// TIA Portal project "TestProject" (V19)

(* hardware
DEVICE "S7-1500/ET200MP station_3"  S7-1500 station
   slot 0: "Rail_0"  Rack  6ES7 590-1***0-0AA0
   slot 1: "PLC_3"  CPU 1511-1 PN  6ES7 511-1AK02-0AB0  V2.8
      slot 3: "CPU display_1"  6ES7591-1AA00-0AA0
      slot 32768: "PROFINET interface_1"  X1
         slot 32769: "Port_1"  X1 P1
         slot 32770: "Port_2"  X1 P2
      slot 34817: "Virtual CP interface port_1"  Virtual CP interface port  Virtual CP interface port
*)

// ===== PLC "PLC_3"  CPU 1511-1 PN =====

DATA_BLOCK "DTLToString_ISO_DB"   // DB1
{ S7_Optimized_Access := 'TRUE' }
VERSION : 0.1
   VAR
      "date" : DTL;
      separator : Char;
      DTLToString_ISO : String;
   END_VAR
BEGIN
END_DATA_BLOCK

DATA_BLOCK "ExtractStringFromCharArray_DB"   // DB2
{ S7_Optimized_Access := 'TRUE' }
VERSION : 0.1
   VAR
      textBefore : String;
      textAfter : String;
      extractedString : String;
      status : Word;
      searchIn : Array[0..9] of Char;
      ExtractStringFromCharArray : Word;
   END_VAR
BEGIN
END_DATA_BLOCK

DATA_BLOCK "MatrixAddition_DB"   // DB3
{ S7_Optimized_Access := 'TRUE' }
VERSION : 0.1
   VAR
      matrix1 : Array[1..2, 1..2] of LReal;
      matrix2 : Array[1..2, 1..2] of LReal;
      error : Bool;
      status : Word;
      matrixResult : Array[1..2, 1..2] of LReal;
   END_VAR
BEGIN
END_DATA_BLOCK

DATA_BLOCK "RandomRange_DInt_DB"   // DB4
{ S7_Optimized_Access := 'TRUE' }
VERSION : 0.1
   VAR
      minValue : DInt;
      maxValue : DInt;
      error : Bool;
      status : Word;
      subfunctionStatus : Word;
      RandomRange_DInt : DInt;
   END_VAR
BEGIN
END_DATA_BLOCK

DATA_BLOCK "SearchMinMax_DInt_DB"   // DB5
{ S7_Optimized_Access := 'TRUE' }
VERSION : 0.1
   VAR
      values : Array[0..9] of DInt;
      minValue : DInt;
      minValueIndex : DInt;
      maxValue : DInt;
      maxValueIndex : DInt;
   END_VAR
BEGIN
END_DATA_BLOCK

DATA_BLOCK "StringToTaddr_DB"   // DB6
{ S7_Optimized_Access := 'TRUE' }
VERSION : 0.1
   VAR
      ipAddressString : String;
      error : Bool;
      status : Word;
      StringToTaddr : TADDR_Param;
   END_VAR
BEGIN
END_DATA_BLOCK

DATA_BLOCK "FIFO_DB"   // DB7
{ S7_Optimized_Access := 'TRUE' }
VERSION : 0.1
// stored: InstanceOfName FIFO
"FIFO"
BEGIN
END_DATA_BLOCK

DATA_BLOCK "FIFO_DBG"   // DB8
{ S7_Optimized_Access := 'TRUE' }
VERSION : 0.1
   VAR
      enqueue : Bool;
      dequeue : Bool;
      reset : Bool;
      clear : Bool;
      initialItem : Int;
      error : Bool;
      status : Word;
      subFunctionStatus : Word;
      elementCount : DInt;
      isEmpty : Bool;
      item : Int;
      buffer : Array[1..3] of Int;
   END_VAR
BEGIN
END_DATA_BLOCK

DATA_BLOCK "FloatingAverage_DB"   // DB9
{ S7_Optimized_Access := 'TRUE' }
VERSION : 0.1
// stored: InstanceOfName FloatingAverage
"FloatingAverage"
BEGIN
END_DATA_BLOCK

DATA_BLOCK "Frequency_DB"   // DB10
{ S7_Optimized_Access := 'TRUE' }
VERSION : 0.1
// stored: InstanceOfName Frequency
"Frequency"
BEGIN
END_DATA_BLOCK

DATA_BLOCK "GetBitStates_DB"   // DB11
{ S7_Optimized_Access := 'TRUE' }
VERSION : 0.1
// stored: InstanceOfName GetBitStates
"GetBitStates"
BEGIN
END_DATA_BLOCK

DATA_BLOCK "Integration_DB"   // DB12
{ S7_Optimized_Access := 'TRUE' }
VERSION : 0.1
// stored: InstanceOfName Integration
"Integration"
BEGIN
END_DATA_BLOCK

DATA_BLOCK "ShellSort_DInt_DB"   // DB13
{ S7_Optimized_Access := 'TRUE' }
VERSION : 0.1
// stored: InstanceOfName ShellSort_DInt
"ShellSort_DInt"
BEGIN
END_DATA_BLOCK

DATA_BLOCK "ShellSort_DInt_DBG"   // DB14
{ S7_Optimized_Access := 'TRUE' }
VERSION : 0.1
   VAR
      sortDirection : Bool;
      error : Bool;
      status : Word;
      "array" : Array[1..5] of DInt;
   END_VAR
BEGIN
END_DATA_BLOCK

DATA_BLOCK "StackMin_DB"   // DB15
{ S7_Optimized_Access := 'TRUE' }
VERSION : 0.1
// stored: InstanceOfName StackMin
"StackMin"
BEGIN
END_DATA_BLOCK

DATA_BLOCK "StackMin_DBG"   // DB16
{ S7_Optimized_Access := 'TRUE' }
VERSION : 0.1
   VAR
      push : Bool;
      pop : Bool;
      reset : Bool;
      error : Bool;
      status : Word;
      item : Int;
      stack : Array[0..3] of Int;
   END_VAR
BEGIN
END_DATA_BLOCK

DATA_BLOCK "TempCtrl_DB"   // DB17
{ S7_Optimized_Access := 'TRUE' }
VERSION : 0.1
// stored: InstanceOfName TempCtrl
"TempCtrl"
BEGIN
END_DATA_BLOCK

DATA_BLOCK "LightsControl_DB"   // DB18
{ S7_Optimized_Access := 'TRUE' }
VERSION : 0.1
// stored: InstanceOfName LightsControl
"LightsControl"
BEGIN
END_DATA_BLOCK

DATA_BLOCK "MatrixAddition_DBG"   // DB19
{ S7_Optimized_Access := 'TRUE' }
VERSION : 0.1
   VAR
      matrix1 : Array[1..4] of LReal;
      matrix2 : Array[1..4] of LReal;
      matrixResult : Array[1..4] of LReal;
   END_VAR
BEGIN
END_DATA_BLOCK

DATA_BLOCK "MatrixMultiplication_DB"   // DB20
{ S7_Optimized_Access := 'TRUE' }
VERSION : 0.1
   VAR
      matrix1 : Array[1..2, 1..2] of LReal;
      matrix2 : Array[1..2, 1..2] of LReal;
      error : Bool;
      status : Word;
      matrixResult : Array[1..2, 1..2] of LReal;
   END_VAR
BEGIN
END_DATA_BLOCK

DATA_BLOCK "MatrixMultiplication_DBG"   // DB21
{ S7_Optimized_Access := 'TRUE' }
VERSION : 0.1
   VAR
      matrix1 : Array[1..4] of LReal;
      matrix2 : Array[1..4] of LReal;
      matrixResult : Array[1..4] of LReal;
   END_VAR
BEGIN
END_DATA_BLOCK

FUNCTION_BLOCK "FIFO"   // FB1, SCL
{ S7_Optimized_Access := 'TRUE' }
   VAR_INPUT
      enqueue : Bool := FALSE;
      dequeue : Bool := FALSE;
      reset : Bool;
      clear : Bool;
      initialItem : Variant;
   END_VAR
   VAR_OUTPUT
      error : Bool;
      status : Word;
      elementCount : DInt := 0;
      isEmpty : Bool := FALSE;
   END_VAR
   VAR_IN_OUT
      item : Variant;
      buffer : Variant;
   END_VAR
   VAR
      statEdgesMem : Struct
         enqueue : Bool;
         dequeue : Bool;
         clear : Bool;
      END_STRUCT;
      statFirstItemIndex : Int := -1;
      statNextEmptyItemIndex : Int := 0;
      statElementCount : DInt;
   END_VAR
   VAR_TEMP
      tempEdges : Struct
         enqueue : Bool;
         dequeue : Bool;
         clear : Bool;
      END_STRUCT;
      tempInternalError : Int;
      tempNewFirstItemIndex : Int;
      tempNewNextEmptyItemIndex : Int;
      tempBufferSize : UDInt;
      tempCounter : Int;
   END_VAR
   VAR CONSTANT
      BUFFER_IS_EMPTY : Int := -1;
      NO_INTERNAL_ERROR : Int := 0;
      BUFFER_INITIALIZED : Int := -1;
      EMPTY_INITIALIZED : Int := 0;
      INDEX_BEGINNING : Int := 0;
      COUNT_ELEMENTS : UDInt := 1;
      INCREMENT : Int := 1;
      BUFFER_SIZE_CORRECTION : UDInt := 1;
      COUNTER_LOWER_LIMIT : Int := 0;
      ZERO_ELEMENTS : DInt := 0;
      STATUS_NO_ERROR : Word := 16#0000;
      STATUS_NO_CURRENT_JOBS : Word := 16#7000;
      ERR_BUFFER_EMPTY : Word := 16#8001;
      ERR_BUFFER_FULL : Word := 16#8002;
      ERR_NO_ARRAY : Word := 16#8200;
      ERR_WRONG_TYPE_ITEM : Word := 16#8201;
      ERR_WRONG_TYPE_INITIAL_ITEM : Word := 16#8202;
      ERR_INDEX_IN_ARRAY_LIMITS_1 : Word := 16#8601;
      ERR_INDEX_IN_ARRAY_LIMITS_2 : Word := 16#8602;
      ERR_CLEAR_BUFFER : Word := 16#8610;
      ERR_RETURN_FIRST_ENTRY : Word := 16#8611;
      ERR_REPLACE_ITEM_BY_INIT_VALUE : Word := 16#8612;
      ERR_WRITE_ENTRY : Word := 16#8613;
   END_VAR
BEGIN
   REGION Block info header
       //===============================================================================
       // Title:           FIFO
       // Comment/Function: FIFO (First In First Out)
       //                   Queue / ring buffer memory

       //=============================================================================
   END_REGION Block info header

   REGION Block execution control
       // collect edges
       #tempEdges.enqueue := #enqueue AND NOT #statEdgesMem.enqueue;
       #tempEdges.dequeue := #dequeue AND NOT #statEdgesMem.dequeue;
       #tempEdges.clear := #clear AND NOT #statEdgesMem.clear;
       // store values for edge detection
       #statEdgesMem.enqueue := #enqueue;
       #statEdgesMem.dequeue := #dequeue;
       #statEdgesMem.clear := #clear;

       // This program code section is only executed if no trigger input is active
       IF NOT (#enqueue OR #dequeue OR #reset OR #clear) THEN
           // If an error occurred during program execution,
           // the status "No Current Job" is used 16#7000 afterwarts when the triggers are reseted
           #error := false;
           #status := #STATUS_NO_CURRENT_JOBS;

           // the program processing OF the FB is terminated
           RETURN;
       END_IF;
   END_REGION

   REGION Validation of inputs
       // check whether the ring #buffer is an ARRAY.
       // IF so, the number OF the ARRAY elements is read out.
       // IF it is NOT an ARRAY, the program execution is terminated at this point
       IF IS_ARRAY(#buffer) THEN
           #tempBufferSize := CountOfElements(#buffer);
       ELSE
           #error := true;
           #status := #ERR_NO_ARRAY;

           RETURN;
       END_IF;

       // check whether the data type OF the ARRAY elements matches
       // the data type OF the entry (#item). IF the data types DO NOT match,
       // the program execution is terminated at this point
       IF (TypeOf(#item) <> TypeOfElements(#buffer)) THEN
           #error := true;
           #status := #ERR_WRONG_TYPE_ITEM;

           RETURN;
       END_IF;

       // check whether the initial value OF the ring #buffer
       // matches the entry (tag #item). IF the data types DO NOT match,
       // the program execution is terminated at this point
       IF (TypeOf(#item) <> TypeOf(#initialItem)) THEN
           #error := true;
           #status := #ERR_WRONG_TYPE_INITIAL_ITEM;

           RETURN;
       END_IF;

       // check whether the variable indices are within the ARRAY limits.
       // IF they are NOT, the program execution is terminated at this point
       IF (#statNextEmptyItemIndex >= #tempBufferSize) THEN
           #error := true;
           #status := #ERR_INDEX_IN_ARRAY_LIMITS_1;

           RETURN;
       ELSIF (#statFirstItemIndex >= #tempBufferSize) THEN
           #error := true;
           #status := #ERR_INDEX_IN_ARRAY_LIMITS_2;

           RETURN;
       END_IF;

       // If resetBuffer is "TRUE", the buffer counters are reset
       IF #reset THEN
           #statFirstItemIndex := #BUFFER_INITIALIZED;
           #statNextEmptyItemIndex := #EMPTY_INITIALIZED;
           #statElementCount := #EMPTY_INITIALIZED;
           #elementCount := #EMPTY_INITIALIZED;
           #isEmpty := true;
           RETURN;
       END_IF;

       // If clearBuffer has rising edge, the buffer is initialized by initial values
       IF #tempEdges.clear THEN
           FOR #tempCounter := #COUNTER_LOWER_LIMIT TO UDINT_TO_INT(#tempBufferSize - #BUFFER_SIZE_CORRECTION) DO

               #tempInternalError := MOVE_BLK_VARIANT(SRC := #initialItem,
                                                      COUNT := #COUNT_ELEMENTS,
                                                      SRC_INDEX := #INDEX_BEGINNING,
                                                      DEST_INDEX := #tempCounter,
                                                      DEST => #buffer);
           END_FOR;

           // checks whether a local error has occurred.
           IF (#tempInternalError <> #NO_INTERNAL_ERROR) THEN
               #error := true;
               #status := #ERR_CLEAR_BUFFER;

           END_IF;

           // reset counters
           #statFirstItemIndex := #BUFFER_INITIALIZED;
           #statNextEmptyItemIndex := #EMPTY_INITIALIZED;
           #statElementCount := #EMPTY_INITIALIZED;
           #elementCount := #EMPTY_INITIALIZED;
           #isEmpty := true;
           RETURN;
       END_IF;
   END_REGION

   REGION FIFO algorithm  
       IF #tempEdges.dequeue THEN
           REGION dequeue
               // check whether the ring #buffer is empty
               // IF this is the CASE, program execution is terminated at this point
               IF (#statFirstItemIndex = #BUFFER_IS_EMPTY) THEN
                   #error := true;
                   #status := #ERR_BUFFER_EMPTY;

                   RETURN;
               END_IF;

               // return the first entry of the ring buffer
               #tempInternalError := MOVE_BLK_VARIANT(SRC := #buffer,
                                                      COUNT := #COUNT_ELEMENTS,
                                                      SRC_INDEX := #statFirstItemIndex,
                                                      DEST_INDEX := #INDEX_BEGINNING,
                                                      DEST => #item);

               // check whether a local error has occurred
               IF (#tempInternalError <> #NO_INTERNAL_ERROR) THEN
                   #error := true;
                   #status := #ERR_RETURN_FIRST_ENTRY;

                   RETURN;
               END_IF;

               // check whether the ring #buffer contains ARRAY elements
               // IF it does, the first entry is passed further on and the index is incremented BY 1
               #tempInternalError := MOVE_BLK_VARIANT(SRC := #initialItem,
                                                      COUNT := #COUNT_ELEMENTS,
                                                      SRC_INDEX := #INDEX_BEGINNING,
                                                      DEST_INDEX := #statFirstItemIndex,
                                                      DEST => #buffer);

               // check whether a local error has occurred
               IF (#tempInternalError <> #NO_INTERNAL_ERROR) THEN
                   #error := true;
                   #status := #ERR_REPLACE_ITEM_BY_INIT_VALUE;

                   RETURN;
               END_IF;

               // calculate the new index of the first entry
               #tempNewFirstItemIndex := #statFirstItemIndex + #INCREMENT;
               #tempNewFirstItemIndex := #tempNewFirstItemIndex MOD UDINT_TO_INT(#tempBufferSize);

               // check whether the ring buffer is empty
               IF (#statNextEmptyItemIndex = #tempNewFirstItemIndex) THEN
                   // If the ring buffer is empty, the index is set to 0
                   #statFirstItemIndex := #BUFFER_INITIALIZED;
                   #statNextEmptyItemIndex := #EMPTY_INITIALIZED;
               ELSE
                   // The index of the first entry is changed
                   #statFirstItemIndex := #tempNewFirstItemIndex;
               END_IF;

               // Evaluation of the number of elements in the stack
               #statElementCount -= #INCREMENT;

           END_REGION dequeue

       ELSIF #tempEdges.enqueue THEN
           REGION enqueue
               // check whether the ring #buffer is full
               // IF this is the CASE, program execution is terminated at this point
               IF (#statNextEmptyItemIndex = #statFirstItemIndex) THEN
                   #error := true;
                   #status := #ERR_BUFFER_FULL;

                   RETURN;
               END_IF;

               // write the entry to the ring buffer
               #tempInternalError := MOVE_BLK_VARIANT(SRC := #item,
                                                      COUNT := #COUNT_ELEMENTS,
                                                      SRC_INDEX := #INDEX_BEGINNING,
                                                      DEST_INDEX := #statNextEmptyItemIndex,
                                                      DEST => #buffer);

               // check whether a local error has occurred
               IF (#tempInternalError <> #NO_INTERNAL_ERROR) THEN
                   #error := true;
                   #status := #ERR_WRITE_ENTRY;

                   RETURN;
               END_IF;

               // increment the index by 1 and calculates the new empty entry index
               #tempNewNextEmptyItemIndex := (#statNextEmptyItemIndex + #INCREMENT) MOD UDINT_TO_INT(#tempBufferSize);
               #statNextEmptyItemIndex := #tempNewNextEmptyItemIndex;

               // check which index the "#firstItemIndex" tag has
               // IF the number = -1, the ring buffer is initialized
               // AND the entry is written TO the ring #buffer
               // Therefore, "0" must be assigned TO the tag
               IF (#statFirstItemIndex = #BUFFER_INITIALIZED) THEN
                   #statFirstItemIndex := #INDEX_BEGINNING;
               END_IF;

               // Evaluation of the number of elements in the stack
               #statElementCount += #INCREMENT;
           END_REGION enqueue
       END_IF;
   END_REGION

   REGION Writing to outputs
       #elementCount := #statElementCount;
       #isEmpty := #statElementCount <= #ZERO_ELEMENTS;

       #error := false;
       #status := #STATUS_NO_ERROR;

       // no error handling by ENO needed
       ENO := TRUE;
   END_REGION
END_FUNCTION_BLOCK

FUNCTION_BLOCK "FloatingAverage"   // FB2, SCL
{ S7_Optimized_Access := 'TRUE' }
   VAR_INPUT
      cyclicExecution : Bool := FALSE;
      trigger : Bool;
      value : LReal;
      windowSize : Int := 100;
      reset : Bool;
   END_VAR
   VAR_OUTPUT
      average : LReal;
      windowSizeReached : Bool;
      error : Bool;
      status : Word;
   END_VAR
   VAR
      statValues : Array[#ZERO_INT..#MAX_WINDOW_SIZE] of LReal;
      statValuesSum : LReal := 0.0;
      statArithmeticAverage : LReal := 0.0;
      statWindowSizeOld : Int := 0;
      statCounter : Int := 0;
      statwindowSizeReached : Bool;
      statTriggerOld : Bool := FALSE;
   END_VAR
   VAR_TEMP
      tempValue : LReal;
      tempIndex : Int;
      tempTriggerEdge : Bool;
   END_VAR
   VAR CONSTANT
      ZERO_INT : Int := 0;
      ZERO_LREAL : LReal := 0.0;
      MAX_WINDOW_SIZE : Int := 100;
      INCREMENT : Int := 1;
      STATUS_FINISHED_NO_ERROR : Word := 16#0000;
      ERR_WRONG_WINDOW_SIZE : Word := 16#8200;
   END_VAR
BEGIN
   REGION Block info header
       //===============================================================================
       // Title:            FloatingAverage
       // Comment/Function: This function block calculates the floating arithmetic average
       //                   of incoming REAL values each cycle or each trigger impulse.

       //=============================================================================
   END_REGION Block info header

   REGION DESCRIPTION
       (/**/)
   END_REGION DESCRIPTION

   REGION Initialization and input data processing
       // Copy commonly used data to temp variables
       #tempValue := #value;

       // Positive edge detection for triggering of calculation
       #tempTriggerEdge := #trigger AND NOT #statTriggerOld;
       #statTriggerOld := #trigger;

       // Reset OR if window size changes the calculation
       IF #reset OR (#windowSize <> #statWindowSizeOld) THEN
           #statWindowSizeOld := #windowSize;
           #statCounter := #ZERO_INT;
           #statValuesSum := #ZERO_LREAL;
           #statArithmeticAverage := #ZERO_LREAL;
           #average := #ZERO_LREAL;
           #windowSizeReached := FALSE;
           #statwindowSizeReached := FALSE;
           #error := false;
           #status := #STATUS_FINISHED_NO_ERROR;
           RETURN;

           // Check window size, in case of incorrect window size setup an error
       ELSIF (#windowSize <= #ZERO_INT) OR (#windowSize > #MAX_WINDOW_SIZE) THEN
           #statWindowSizeOld := #windowSize;
           #statCounter := #ZERO_INT;
           #statValuesSum := #ZERO_LREAL;
           #statArithmeticAverage := #ZERO_LREAL;
           #average := #ZERO_LREAL;
           #statwindowSizeReached := FALSE;
           #windowSizeReached := FALSE;
           #error := TRUE;
           #status := #ERR_WRONG_WINDOW_SIZE; // Info "No correct set of window size"
           RETURN;
       END_IF;
   END_REGION

   REGION Floating average calculation
       // Triggered calculation OR cyclicly operation
       IF #cyclicExecution OR #tempTriggerEdge THEN

           //Calculate array counter by using modulo
           #tempIndex := #statCounter MOD #windowSize;

           // First step - fill the Array with values
           // as long as desired window size is not reached
           // counter and array starts with zero
           IF (#statCounter < #windowSize) THEN
               // Add value to sum
               #statValuesSum += #tempValue;
               // Add value to window
               #statValues[#tempIndex] := #tempValue;
               // Increment counter
               #statCounter += #INCREMENT;
               // Calculate avarage value
               #statArithmeticAverage := #statValuesSum / #statCounter;

           ELSE
               // wuindow size is reached, set output
               #statwindowSizeReached := TRUE;
               // Add value to sum
               #statValuesSum += #tempValue - #statValues[#tempIndex];
               // Add value to window
               #statValues[#tempIndex] := #tempValue;
               // Calculate avarage value
               #statArithmeticAverage := #statValuesSum / #windowSize;

               // Manipulate counter value of window if modulo calc result is zero
               IF (#tempIndex = #ZERO_INT) THEN
                   #statCounter := #windowSize + #INCREMENT;
               ELSE
                   // Increment counter
                   #statCounter += #INCREMENT;
               END_IF;
           END_IF;
       END_IF;
   END_REGION

   REGION Outputs
       #average := #statArithmeticAverage;
       #windowSizeReached := #statwindowSizeReached;
       #error := FALSE;
       #status := #STATUS_FINISHED_NO_ERROR;

       // ENO mechanism is not used - forced to true
       ENO := TRUE;
   END_REGION
END_FUNCTION_BLOCK

FUNCTION_BLOCK "Frequency"   // FB3, SCL
{ S7_Optimized_Access := 'TRUE' }
   VAR_INPUT
      frequency : Real := 0.0;
      pulsePauseRatio : Real := 1.0;
   END_VAR
   VAR_OUTPUT
      clock : Bool;
      countdown : Time;
   END_VAR
   VAR
      instTofTimePulse : TOF_TIME;
      instTofTimePause : TOF_TIME;
      statFrequencyOld : Real;
      statPulsePauseRatioOld : Real;
      statTimePulse : Time;
      statTimePause : Time;
   END_VAR
   VAR_TEMP
      tempPulseRate : Real;
      tempPauseRate : Real;
      tempCountdown : Time;
   END_VAR
   VAR CONSTANT
      ZERO : Real := 0.0;
      ZERO_TIME : Time := T#0MS;
      SECOND_IN_MS : Real := 1000.0;
      ONE : Real := 1.0;
   END_VAR
BEGIN
   REGION Block info header
       //=============================================================================
       // Title:            Frequency
       // Comment/Function: This function generates a signal that changes between the values `FALSE` and `TRUE` depending on a defined frequency and a pulse pause ratio.

       //=============================================================================
   END_REGION Block info header

   REGION Calculation of settings and program execution
       // If input <= 0.0 the block is disabled
       IF (#frequency <= #ZERO) OR (#pulsePauseRatio <= #ZERO) THEN
           #clock := FALSE;
           #tempCountdown := #ZERO_TIME;
       ELSE

           //Calculating function frequency and pulse pause ratio only when an input is changed
           IF #statFrequencyOld <> #frequency OR #statPulsePauseRatioOld <> #pulsePauseRatio THEN
               RESET_TIMER(TIMER := #instTofTimePause);
               RESET_TIMER(TIMER := #instTofTimePulse);

               #tempPulseRate := #pulsePauseRatio / (#pulsePauseRatio + #ONE); // Calculate pulse rate   
               #tempPauseRate := #ONE - #tempPulseRate;                      // Calculate pause rate   
               #statTimePulse := UDINT_TO_TIME(REAL_TO_UDINT((#SECOND_IN_MS * #tempPulseRate / #frequency))); // Calculate pulse time   
               #statTimePause := UDINT_TO_TIME(REAL_TO_UDINT((#SECOND_IN_MS * #tempPauseRate / #frequency))); // Calculate pause time
               #statFrequencyOld := #frequency;
               #statPulsePauseRatioOld := #pulsePauseRatio;
           END_IF;

           //Two time off-delay timers that are resetting each other on expiration
           #instTofTimePulse(IN := NOT #instTofTimePause.Q,
                             PT := #statTimePulse);

           //If timer for pulse is running, remaining time of the PULSE is calculated
           #tempCountdown := #statTimePulse - #instTofTimePulse.ET;

           #instTofTimePause(IN := #instTofTimePulse.Q,
                             PT := #statTimePause);

           //If timer for pulse is NOT running, remaining time of the PAUSE is calculated
           IF #tempCountdown = #ZERO_TIME THEN
               #tempCountdown := #statTimePause - #instTofTimePause.ET;
           END_IF;

       END_IF;
   END_REGION

   REGION Writing to outputs
       // Assigning value of the pulse timer to the clock output
       #clock := #instTofTimePulse.Q;
       #countdown := #tempCountdown;
       //ENO mechanism is not used - forced to true.
       ENO := TRUE;
   END_REGION
END_FUNCTION_BLOCK

FUNCTION_BLOCK "GetBitStates"   // FB4, SCL
{ S7_Optimized_Access := 'TRUE' }
   VAR_INPUT
      value : DWord;
   END_VAR
   VAR_OUTPUT
      hasChanged : Bool;
      hasRisingEdges : Bool;
      risingBits : DWord;
      noOfRisingBits : USInt;
      hasFallingEdges : Bool;
      fallingBits : DWord;
      noOfFallingBits : USInt;
   END_VAR
   VAR
      statPreviousValue : DWord;
   END_VAR
   VAR_TEMP
      tempRisingResult : DWord;
      tempNoRisingBits : DWord;
      tempFallingResult : DWord;
      tempNoFallingBits : DWord;
   END_VAR
   VAR CONSTANT
      ZERO_EDGES : DWord;
   END_VAR
BEGIN
   REGION BLOCK INFO HEADER
       //============================================================================
       // Title:            GetBitStates
       // Comment/Function: Check DWord for edges, falling as well as rising.  
       //                   Returns the number of edges, DWords with edge bits and a bool if edge(s) exists.
       //                   https://graphics.stanford.edu/~seander/bithacks.html#CountBitsSetParallel

       //=============================================================================
   END_REGION BLOCK INFO HEADER

   REGION PROGRAM LOGIC
       // Get edges from input DWord and DWord from previous cycle
       #tempRisingResult := #value AND NOT #statPreviousValue;
       #tempFallingResult := NOT #value AND #statPreviousValue;

       // Store value for next cycle
       #statPreviousValue := #value;

       // Copy edge result into work variable for counting the number of rising edges
       #tempNoRisingBits := #tempRisingResult;
       // Count number of rising edges, algorythm descriped from: https://graphics.stanford.edu/~seander/bithacks.html#CountBitsSetParallel
       #tempNoRisingBits := UDINT_TO_DWORD(DWORD_TO_UDINT(#tempNoRisingBits) - DWORD_TO_UDINT(SHR(IN := #tempNoRisingBits, N := 1) AND 16#55555555));
       #tempNoRisingBits := UDINT_TO_DWORD(DWORD_TO_UDINT(#tempNoRisingBits & 16#33333333) + DWORD_TO_UDINT(SHR(IN := #tempNoRisingBits, N := 2) AND 16#33333333));
       #tempNoRisingBits := SHR(IN := UDINT_TO_DWORD(DWORD_TO_UDINT(UDINT_TO_DWORD(DWORD_TO_UDINT(#tempNoRisingBits) + DWORD_TO_UDINT(SHR(IN := #tempNoRisingBits, N := 4))) AND 16#0F0F0F0F) * DWORD_TO_UDINT(16#01010101)), N := 24);

       // Copy edges result into work variable for counting the number of falling edges
       #tempNoFallingBits := #tempFallingResult;
       // Count number of falling edges, algorythm descriped from: https://graphics.stanford.edu/~seander/bithacks.html#CountBitsSetParallel
       #tempNoFallingBits := UDINT_TO_DWORD(DWORD_TO_UDINT(#tempNoFallingBits) - DWORD_TO_UDINT(SHR(IN := #tempNoFallingBits, N := 1) AND 16#55555555));
       #tempNoFallingBits := UDINT_TO_DWORD(DWORD_TO_UDINT(#tempNoFallingBits & 16#33333333) + DWORD_TO_UDINT(SHR(IN := #tempNoFallingBits, N := 2) AND 16#33333333));
       #tempNoFallingBits := SHR(IN := UDINT_TO_DWORD(DWORD_TO_UDINT(UDINT_TO_DWORD(DWORD_TO_UDINT(#tempNoFallingBits) + DWORD_TO_UDINT(SHR(IN := #tempNoFallingBits, N := 4))) AND 16#0F0F0F0F) * DWORD_TO_UDINT(16#01010101)), N := 24);
   END_REGION PROGRAM LOGIC

   REGION OUTPUTS
       #hasChanged := (#tempRisingResult > #ZERO_EDGES) OR (#tempFallingResult > #ZERO_EDGES);
       #hasRisingEdges := #tempRisingResult > #ZERO_EDGES;
       #risingBits := #tempRisingResult;
       #noOfRisingBits := DWORD_TO_USINT(#tempNoRisingBits);

       #hasFallingEdges := #tempFallingResult > #ZERO_EDGES;
       #fallingBits := #tempFallingResult;
       #noOfFallingBits := DWORD_TO_USINT(#tempNoFallingBits);

       // ENO not needed, no error evaluation needed
       ENO := FALSE;
   END_REGION OUTPUTS
END_FUNCTION_BLOCK

FUNCTION_BLOCK "Integration"   // FB5, SCL
{ S7_Optimized_Access := 'TRUE' }
   VAR_INPUT
      enable : Bool;
      value : LReal;
      reset : Bool;
   END_VAR
   VAR_OUTPUT
      integral : LReal;
      error : Bool;
      status : Word;
   END_VAR
   VAR
      statLastTime : DTL;
      statInputOldValue : LReal;
      statIntegral : LReal;
   END_VAR
   VAR_TEMP
      tempSysTime : DTL;
      tempTimeDiffrence : LReal;
      tempCalculation : LReal;
      tempRetval : Word;
   END_VAR
   VAR CONSTANT
      CLEAR_TIME : DTL;
      SECOND_IN_MS : LReal := 1000.0;
      DIVIDE_BY_TWO : LReal := 2.0;
      ZERO : LReal := 0.0;
      STATUS_EXECUTION_FINISHED_NO_ERROR : Word := 16#0000;
      SUB_STATUS_NO_ERROR : Word := 16#0000;
      ERR_READ_SYS_TIME : Word := 16#8600;
   END_VAR
BEGIN
   REGION Block info header
       //============================================================================
       // Title:            Integration
       // Comment/Function: Integrates the input value
       //                   integration by trapezoidal rule

       //=============================================================================
   END_REGION Block info header

   //Reset region must be before the enable region so that even if the function disabled, the user can reset the values.
   REGION Reset the function
       IF #reset THEN
           #statInputOldValue := #ZERO;
           #statIntegral := #ZERO;

           // Clear LastTime value.
           // Initial condition - first Delta time will be 0.
           #statLastTime := #CLEAR_TIME;

           #integral := #ZERO;
           #error := false;
           #status := #STATUS_EXECUTION_FINISHED_NO_ERROR;

           RETURN;
       END_IF;
   END_REGION Reset the function

   REGION Enable/Disable integral calculation
       IF NOT #enable THEN
           #statInputOldValue := #ZERO;

           // Clear LastTime value.
           // If it is not cleared when the function is enabled again,
           // the first value will be multiplied with the time difference of the whole disable time
           // Initial condition - first Delta time will be 0.
           #statLastTime := #CLEAR_TIME;

           #integral := #statIntegral;
           #error := false;
           #status := #STATUS_EXECUTION_FINISHED_NO_ERROR;

           RETURN;
       END_IF;
   END_REGION Enable/Disable integral calculation

   REGION Get system time
       // Read system time
       #tempRetval := INT_TO_WORD(RD_SYS_T(OUT => #tempSysTime));

       // Error Handling read system time
       IF (#tempRetval > #SUB_STATUS_NO_ERROR) THEN
           #integral := #statIntegral;
           #error := TRUE;
           #status := #ERR_READ_SYS_TIME;

           RETURN;
       END_IF;
   END_REGION

   REGION Calculating the integral
       // Calculate time difference between last and actual time
       // coverting from DTL via time and DInt to Real
       // scale from millisecond to second
       #tempTimeDiffrence := DINT_TO_REAL(TIME_TO_DINT(T_DIFF(IN1 := #tempSysTime, IN2 := #statLastTime))) / #SECOND_IN_MS;

       // Write actual to last time
       #statLastTime := #tempSysTime;

       // integration by trapezoidal rule
       // add LastScalIn to ScalIn
       // divide by two --> avarage of both - old and actual value
       // multiply with time delta --> area unterneath the both borders
       #tempCalculation := (#value + #statInputOldValue) * #tempTimeDiffrence / #DIVIDE_BY_TWO;

       // Calculate new integral
       #statIntegral += #tempCalculation;

       // Save last input
       #statInputOldValue := #value;
   END_REGION Calculating the integral

   REGION Write outputs
       #integral := #statIntegral;
       #error := false;
       #status := #STATUS_EXECUTION_FINISHED_NO_ERROR;


       //ENO mechanism is not used
       ENO := TRUE;
   END_REGION Write outputs
END_FUNCTION_BLOCK

FUNCTION_BLOCK "ShellSort_DInt"   // FB6, SCL
{ S7_Optimized_Access := 'TRUE' }
   VAR_INPUT
      sortDirection : Bool;
   END_VAR
   VAR_OUTPUT
      error : Bool;
      status : Word;
   END_VAR
   VAR_IN_OUT
      "array" : Array[*] of DInt;
   END_VAR
   VAR
      tempArray : Array[1..#MAX_ARRAY_ELEMENTS] of DInt;
   END_VAR
   VAR_TEMP
      tempLowerLimit : DInt;
      tempUpperLimit : DInt;
      tempNoOfElements : DInt;
      tempGap : DInt;
      tempLoopIndex : DInt;
      tempExchangeIndex : DInt;
      tempExchangeVariable : DInt;
      tempArrayOffset : DInt;
   END_VAR
   VAR CONSTANT
      ARRAY_FIRST_DIMENSION : UInt := 1;
      ARRAY_START_INDEX : UInt := 1;
      SINGLE_ARRAY_ELEMENT : DInt := 1;
      GAP_INIT : Int := 1;
      GAP_THRESHOLD : Int := 1;
      GAP_RATIO : DInt := 3;
      INCREMENT : Int := 1;
      ELEMENTS_COUNT_CORRECTION : DInt := 1;
      MAX_ARRAY_ELEMENTS : Int := 1000;
      STATUS_NO_ERROR : Word := 16#0000;
      ERR_NO_ARRAY : Word := 16#8200;
      ERR_TOO_MANY_ELEMENTS : Word := 16#8201;
   END_VAR
BEGIN
   REGION Block info header
       //===============================================================================
       // Title:            ShellSort_DInt
       // Comment/Function: This block sorts an array with any number of elements (max. 1000)
       //                   in ascending or descending order and returns the sorted version of the array in the same variable.

       //=============================================================================
   END_REGION Block info header

   REGION Special description
       // Space note: If you wish to reduce the space of this block, you may reduce the
       // size OF the tempArray<Type> TO one just big enough FOR your specific purpose
       // It is not recommended to increase the size significantly.
   END_REGION

   REGION Initialization and input data processing
       // Input array size calculation
       #tempLowerLimit := LOWER_BOUND(ARR := #array, DIM := #ARRAY_FIRST_DIMENSION);
       #tempUpperLimit := UPPER_BOUND(ARR := #array, DIM := #ARRAY_FIRST_DIMENSION);

       // Array elements calculation
       // (for example: 6 - 2 = 4; but real number of elements is 5)
       #tempNoOfElements := #tempUpperLimit - #tempLowerLimit + #ELEMENTS_COUNT_CORRECTION;

       // Shift array index to range 1..MAX_ARRAY_ELEMENTS
       #tempArrayOffset := - #tempLowerLimit + #ARRAY_START_INDEX;

       // Check whether the array contains less than the maximum possible amount of elements
       IF #tempNoOfElements > #MAX_ARRAY_ELEMENTS THEN
           #error := true;
           #status := #ERR_TOO_MANY_ELEMENTS;
           RETURN;
       ELSIF #tempNoOfElements <= #SINGLE_ARRAY_ELEMENT THEN
           // If there are 0 elements in the array, set status to "Error: Parameter is an empty array"
           #error := true;
           #status := #ERR_NO_ARRAY;
           RETURN;
       END_IF;
   END_REGION

   REGION Sorting
       // Read the elements of the incoming array and write into the local array
       FOR #tempLoopIndex := #tempLowerLimit TO #tempUpperLimit DO
           #tempArray[#tempLoopIndex + #tempArrayOffset] := #array[#tempLoopIndex];
       END_FOR;

       REGION Shell sort algorithm
           #tempGap := #GAP_INIT;

           // Evaluation of the maximal gap size
           REPEAT
               #tempGap := (#GAP_RATIO * #tempGap) + #INCREMENT;
           UNTIL #tempGap > #tempNoOfElements END_REPEAT;

           REPEAT
               #tempGap := #tempGap / #GAP_RATIO;

               FOR #tempLoopIndex := #tempGap + #INCREMENT TO #tempNoOfElements DO
                   #tempExchangeVariable := #tempArray[#tempLoopIndex];
                   #tempExchangeIndex := #tempLoopIndex;

                   // sort descending 
                   IF #sortDirection THEN
                       WHILE ((#tempArray[#tempExchangeIndex - #tempGap] < #tempExchangeVariable)) DO
                           #tempArray[#tempExchangeIndex] := #tempArray[#tempExchangeIndex - #tempGap];
                           #tempExchangeIndex := #tempExchangeIndex - #tempGap;

                           IF (#tempExchangeIndex <= #tempGap) THEN
                               EXIT;
                           END_IF;
                       END_WHILE;

                       // sort ascending
                   ELSE
                       WHILE ((#tempArray[#tempExchangeIndex - #tempGap] > #tempExchangeVariable)) DO
                           #tempArray[#tempExchangeIndex] := #tempArray[#tempExchangeIndex - #tempGap];
                           #tempExchangeIndex := #tempExchangeIndex - #tempGap;

                           IF (#tempExchangeIndex <= #tempGap) THEN
                               EXIT;
                           END_IF;
                       END_WHILE;
                   END_IF;

                   #tempArray[#tempExchangeIndex] := #tempExchangeVariable;
               END_FOR;

           UNTIL #tempGap <= #GAP_THRESHOLD END_REPEAT;
       END_REGION

       // Write the elements of the local array back to the inOut array
       FOR #tempLoopIndex := #tempLowerLimit TO #tempUpperLimit DO
           #array[#tempLoopIndex] := #tempArray[#tempLoopIndex + #tempArrayOffset];
       END_FOR;

       // Set "No error" status
       #error := false;
       #status := #STATUS_NO_ERROR;

       // no error handling needed
       ENO := TRUE;
   END_REGION
END_FUNCTION_BLOCK

FUNCTION_BLOCK "StackMin"   // FB7, SCL
{ S7_Optimized_Access := 'TRUE' }
   VAR_INPUT
      push : Bool;   // 入栈
      pop : Bool;   // 出栈
      reset : Bool;   // 复位
   END_VAR
   VAR_OUTPUT
      error : Bool;   // 故障状态
      status : Word;   // 状态代码
   END_VAR
   VAR_IN_OUT
      item : Int;   // 入栈或出栈的元素
      stack : Array[0..3] of Int;   // 堆栈空间
   END_VAR
   VAR
      statStackIndex : Int;   // 堆栈指针
      statMin : Int;
   END_VAR
   VAR_TEMP
      tempStackSize : DInt;
      tempCount : Int;
   END_VAR
   VAR CONSTANT
      STACK_FULL : Word := 16#8A04;   // 堆栈已满
      STACK_EMPTY : Word := 16#8A05;   // 堆栈已空
      NO_ERROR : Word := 16#0000;
   END_VAR
BEGIN
   //设置堆栈长度
   REGION StackSize
       #tempStackSize := 4;
   END_REGION

   //入栈
   REGION Push
       IF #push = TRUE THEN
           IF #statStackIndex >= #tempStackSize THEN             //判断是否满栈，如果已经满栈,则不执行入栈,并报错
               #error := TRUE;
               #status := #STACK_FULL;
               RETURN;
           END_IF;
           #stack[#statStackIndex] := #item;                    //否则放入元素
           #statStackIndex += 1;                                //堆栈指针上移
       END_IF;
   END_REGION

   //出栈
   REGION Pop
       IF #pop = TRUE THEN

           //判断空栈，如果已经空栈,则不执行出栈,并报错
           IF #statStackIndex <= 0 THEN
               #error := TRUE;
               #status := #STACK_EMPTY;
               RETURN;
           END_IF;

           //查找最小值所在位置
           #statMin := 0;
           IF #statStackIndex > 1 THEN
               FOR #tempCount := 1 TO #statStackIndex - 1 DO
                   IF #stack[#tempCount] < #stack[#statMin] THEN
                       #statMin := #tempCount;
                   END_IF;
               END_FOR;
           END_IF;

           //取出元素，上面元素往下顺移
           #item := #stack[#statMin];
           IF #statMin <> #statStackIndex - 1 THEN
               FOR #tempCount := #statMin TO #statStackIndex - 2 DO
                   #stack[#tempCount] := #stack[#tempCount + 1];
               END_FOR;
           END_IF;
           #stack[#statStackIndex - 1] := 0;
           #statStackIndex -= 1;                               //堆栈指针下移
       END_IF;
   END_REGION

   //复位
   REGION Reset
       IF #reset = TRUE THEN
           #statStackIndex := 0;
       END_IF;
   END_REGION

   #error := FALSE;
   #status := #NO_ERROR;
END_FUNCTION_BLOCK

FUNCTION_BLOCK "TempCtrl"   // FB8, SCL
{ S7_Optimized_Access := 'TRUE' }
   VAR_INPUT
      TemperatureSensorInput : Real;   // 温度传感器输入值
      SetTemperature : Real;   // 设定温度值
   END_VAR
   VAR_OUTPUT
      CurrentTemperature : Real;   // 当前温度显示
      SetTempDisplay : Real;   // 设定温度显示
      HeaterStatus : Bool;   // 加热器状态显示
      OverheatProtection : Bool;   // 过热保护状态显示
   END_VAR
   VAR_IN_OUT
      HeaterOutput : Bool;   // 加热器控制输出
   END_VAR
   VAR
      HeaterState : Struct
         IsEnabled : Bool;
         OverheatProtectionTriggered : Bool;
      END_STRUCT;
      OverheatTimer : TON_TIME;   // 过热保护定时器
      SensorError : Bool;   // 传感器错误标志
      CoolTimer : TON_TIME;
      OverheatTimerOutput : Bool;
      CoolTimerOutput : Bool;
   END_VAR
BEGIN
   // 显示当前温度和设定温度 
   #CurrentTemperature := #TemperatureSensorInput;
   #SetTempDisplay := #SetTemperature;

   // 检查传感器是否失效 
   IF #TemperatureSensorInput < 0 OR #TemperatureSensorInput > 100 THEN
       #SensorError := TRUE;
   ELSE
       #SensorError := FALSE;
   END_IF;

   // 温度控制逻辑 
   // 过热保护逻辑 
   #OverheatTimer(IN := #HeaterOutput,
                  PT := T#5S,
                  Q => #OverheatTimerOutput);
   IF #HeaterState.IsEnabled AND #OverheatTimerOutput THEN
       #HeaterState.OverheatProtectionTriggered := TRUE;
       #HeaterState.IsEnabled := FALSE;
       #HeaterOutput := FALSE;
   END_IF;
   #CoolTimer(IN := #HeaterState.OverheatProtectionTriggered,
              PT := t#3S,
              Q => #CoolTimerOutput);
   IF #CoolTimerOutput THEN
       #HeaterState.OverheatProtectionTriggered := FALSE;
   END_IF;

   IF NOT #SensorError THEN
       IF #CurrentTemperature < #SetTemperature AND NOT #HeaterState.OverheatProtectionTriggered THEN
           IF NOT #HeaterState.IsEnabled THEN
               #HeaterState.IsEnabled := TRUE;
               #HeaterOutput := TRUE;
           END_IF;
       ELSIF #CurrentTemperature > #SetTemperature THEN
           IF #HeaterState.IsEnabled THEN
               #HeaterState.IsEnabled := FALSE;
               #HeaterOutput := FALSE;
           END_IF;
       END_IF;

   ELSE
       // 传感器错误处理 
       #HeaterOutput := FALSE;
       #HeaterState.IsEnabled := FALSE;
   END_IF;

   // 显示加热器状态和过热保护状态 
   #HeaterStatus := #HeaterState.IsEnabled;
   #OverheatProtection := #HeaterState.OverheatProtectionTriggered;
END_FUNCTION_BLOCK

FUNCTION_BLOCK "LightsControl"   // FB9, SCL
{ S7_Optimized_Access := 'TRUE' }
VERSION : 0.1
   VAR_INPUT
      button1 : Bool;
      button2 : Bool;
      button3 : Bool;
   END_VAR
   VAR_OUTPUT
      greenLight : Bool;
      redLight : Bool;
      yellowLight : Bool;
   END_VAR
   VAR
      CycleStep : Int := 0;
      ManModeTimer1 : TON_TIME;
      ManModeTimer2 : TON_TIME;
      AutoModeTimer : TON_TIME;
   END_VAR
BEGIN
       IF #button1 = FALSE THEN
           #ManModeTimer1(IN := #ManModeTimer2.Q,
                          PT := t#1s);
           #ManModeTimer2(IN := NOT #ManModeTimer1.Q,
                          PT := t#1s);
           IF #button2 AND NOT #button3 THEN
               #greenLight := TRUE;
               #redLight := #ManModeTimer2.Q;
               #yellowLight := FALSE;
           ELSIF NOT #button2 AND #button3 THEN
               #redLight := TRUE;
               #yellowLight := #ManModeTimer2.Q;
               #greenLight := FALSE;
           ELSIF #button2 AND #button3 THEN
               #yellowLight := TRUE;
               #greenLight := #ManModeTimer2.Q;
               #redLight := FALSE;
           ELSE
               #greenLight := FALSE;
               #redLight := FALSE;
               #yellowLight := FALSE;
           END_IF;

       ELSE
           #AutoModeTimer(IN := TRUE,
                          PT := T#1s);
           CASE #CycleStep OF
               0:
                   #greenLight := TRUE;
                   #redLight := FALSE;
                   #yellowLight := FALSE;
                   IF #AutoModeTimer.Q THEN
                       #CycleStep := 1;
                       #AutoModeTimer(IN := FALSE,
                                      PT := T#1s);
                   END_IF;
               1:
                   #greenLight := FALSE;
                   #redLight := TRUE;
                   #yellowLight := FALSE;

                   IF #AutoModeTimer.Q THEN
                       #CycleStep := 2;
                       #AutoModeTimer(IN := FALSE,
                                      PT := T#1s);
                   END_IF;
               2:
                   #greenLight := FALSE;
                   #redLight := FALSE;
                   #yellowLight := TRUE;

                   IF #AutoModeTimer.Q THEN
                       #CycleStep := 0;
                       #AutoModeTimer(IN := FALSE,
                                      PT := T#1s);
                   END_IF;
           END_CASE;
       END_IF;
END_FUNCTION_BLOCK

FUNCTION "DTLToString_ISO" : String   // FC1, SCL
{ S7_Optimized_Access := 'TRUE' }
   VAR_INPUT
      "date" : DTL;
      separator : Char;
   END_VAR
   VAR_TEMP
      tempString : String;
      tempIndex : DInt;
   END_VAR
   VAR CONSTANT
      CONVERT_SIZE_YEAR : USInt := 4;
      CONVERT_SIZE_MONTH_DAY_HOUR_MINUTE_SECOND : USInt := 2;
      CONVERT_SIZE_NANOSECOND : USInt := 9;
      CONVERT_PRECISION : USInt := 0;
      CONVERT_FORMAT_TO_STRING : Word := 16#0000;
      CONVERT_START_POSITION_YEAR : UInt := 1;
      CONVERT_START_POSITION_MONTH : UInt := 6;
      CONVERT_START_POSITION_DAY : UInt := 9;
      CONVERT_START_POSITION_HOUR : UInt := 12;
      CONVERT_START_POSITION_MINUTE : UInt := 15;
      CONVERT_START_POSITION_SECOND : UInt := 18;
      CONVERT_START_POSITION_NANOSECOND : UInt := 21;
      SEPARATOR_POSITION_YEAR_MONTH : UInt := 5;
      SEPARATOR_POSITION_MONTH_DAY : UInt := 8;
      SEPARATOR_POSITION_HOUR_MINUTE : UInt := 14;
      SEPARATOR_POSITION_MINUTE_SECOND : UInt := 17;
      SEPARATOR_POSITION_SECOND_NANOSECOND : UInt := 20;
      SEPARATOR_NANOSECOND : Char := '.';
      SEPARATOR_TIME : Char := ':';
      SEPARATOR_DATE : Char := '-';
      REPLACE_NANOSECOND_COUNT : DInt := 8;
   END_VAR
BEGIN
   REGION BLOCK INFO HEADER
       //===============================================================================
       // Title:            DTLtoString_ISO
       // Comment/Function: This function converts a date of data type DTL into a character string of data type STRING in international format (YYYY MM DD…).

       //=============================================================================
   END_REGION Block info header

   REGION DESCRIPTION
       (/**/)
   END_REGION DESCRIPTION

   REGION INITIALISATION
       #tempString := '';
   END_REGION

   REGION CONVERTER
       // Set format parameters for output string
       // International ISO 8601
       // DTL  | Y| Y| Y| Y| -| M| M| -| D| D|  | H| H| :| M| M| :| S| S| .|NS|NS|NS|NS|NS|NS|NS|NS|NS
       // -----|--|--|--|--|--|--|--|--|--|--|--|--|--|--|--|--|--|--|--|--|--|--|--|--|--|--|--|--|--
       // Pos  | 1| 2| 3| 4| 5| 6| 7| 8| 9|10|11|12|13|14|15|16|17|18|19|20|21|22|23|24|25|26|27|28|29

       // Convert "Value" into "String" and place at the right position
       VAL_STRG(FORMAT := #CONVERT_FORMAT_TO_STRING,
                IN := #date.YEAR,
                P := #CONVERT_START_POSITION_YEAR,
                PREC := #CONVERT_PRECISION,
                SIZE := #CONVERT_SIZE_YEAR,
                OUT => #tempString);    // DTL YEAR --> String --> #tempPosYear

       VAL_STRG(FORMAT := #CONVERT_FORMAT_TO_STRING,
                IN := #date.MONTH,
                P := #CONVERT_START_POSITION_MONTH,
                PREC := #CONVERT_PRECISION,
                SIZE := #CONVERT_SIZE_MONTH_DAY_HOUR_MINUTE_SECOND,
                OUT => #tempString);     // DTL MONTH --> String --> #tempPosMonth

       VAL_STRG(FORMAT := #CONVERT_FORMAT_TO_STRING,
                IN := #date.DAY,
                P := #CONVERT_START_POSITION_DAY,
                PREC := #CONVERT_PRECISION,
                SIZE := #CONVERT_SIZE_MONTH_DAY_HOUR_MINUTE_SECOND,
                OUT => #tempString);     // DTL DAY --> String --> #tempPosDay

       VAL_STRG(FORMAT := #CONVERT_FORMAT_TO_STRING,
                IN := #date.HOUR,
                P := #CONVERT_START_POSITION_HOUR,
                PREC := #CONVERT_PRECISION,
                SIZE := #CONVERT_SIZE_MONTH_DAY_HOUR_MINUTE_SECOND,
                OUT => #tempString);     // DTL HOUR --> String --> #tempPosHour

       VAL_STRG(FORMAT := #CONVERT_FORMAT_TO_STRING,
                IN := #date.MINUTE,
                P := #CONVERT_START_POSITION_MINUTE,
                PREC := #CONVERT_PRECISION,
                SIZE := #CONVERT_SIZE_MONTH_DAY_HOUR_MINUTE_SECOND,
                OUT => #tempString);     // DTL MINUTE --> String --> #tempPosMinute

       VAL_STRG(FORMAT := #CONVERT_FORMAT_TO_STRING,
                IN := #date.SECOND,
                P := #CONVERT_START_POSITION_SECOND,
                PREC := #CONVERT_PRECISION,
                SIZE := #CONVERT_SIZE_MONTH_DAY_HOUR_MINUTE_SECOND,
                OUT => #tempString);     // DTL SECOND --> String --> #tempPosSecond

       VAL_STRG(FORMAT := #CONVERT_FORMAT_TO_STRING,
                IN := #date.NANOSECOND,
                P := #CONVERT_START_POSITION_NANOSECOND,
                PREC := #CONVERT_PRECISION,
                SIZE := #CONVERT_SIZE_NANOSECOND,
                OUT => #tempString);     // DTL NANOSECOND --> String --> #tempPosNanosecond

       // Place separators at the right position in the string
       IF #separator = '' THEN
           #tempString[#SEPARATOR_POSITION_YEAR_MONTH] := #SEPARATOR_DATE;
           #tempString[#SEPARATOR_POSITION_MONTH_DAY] := #SEPARATOR_DATE;
       ELSE
           #tempString[#SEPARATOR_POSITION_YEAR_MONTH] := #separator;
           #tempString[#SEPARATOR_POSITION_MONTH_DAY] := #separator;
       END_IF;
       #tempString[#SEPARATOR_POSITION_HOUR_MINUTE] := #SEPARATOR_TIME;
       #tempString[#SEPARATOR_POSITION_MINUTE_SECOND] := #SEPARATOR_TIME;
       #tempString[#SEPARATOR_POSITION_SECOND_NANOSECOND] := #SEPARATOR_NANOSECOND;

       // Correcting the string, due to the conversion of a leading "0" value into a "blank".
       // Replacing of "blank" by "0"
       IF (#tempString[#CONVERT_START_POSITION_MONTH] = ' ') THEN
           #tempString[#CONVERT_START_POSITION_MONTH] := '0';
       END_IF;

       IF (#tempString[#CONVERT_START_POSITION_DAY] = ' ') THEN
           #tempString[#CONVERT_START_POSITION_DAY] := '0';
       END_IF;

       IF (#tempString[#CONVERT_START_POSITION_HOUR] = ' ') THEN
           #tempString[#CONVERT_START_POSITION_HOUR] := '0';
       END_IF;

       IF (#tempString[#CONVERT_START_POSITION_MINUTE] = ' ') THEN
           #tempString[#CONVERT_START_POSITION_MINUTE] := '0';
       END_IF;

       IF (#tempString[#CONVERT_START_POSITION_SECOND] = ' ') THEN
           #tempString[#CONVERT_START_POSITION_SECOND] := '0';
       END_IF;

       FOR #tempIndex := 0 TO #REPLACE_NANOSECOND_COUNT DO
           IF (#tempString[UINT_TO_SINT(#CONVERT_START_POSITION_NANOSECOND) + #tempIndex] = ' ') THEN
               #tempString[UINT_TO_SINT(#CONVERT_START_POSITION_NANOSECOND) + #tempIndex] := '0';
           ELSE
               EXIT;
           END_IF;
       END_FOR;
   END_REGION

   REGION OUTPUTS
       #DTLToString_ISO := #tempString;
       // no error handling needed
       ENO := TRUE;
   END_REGION
END_FUNCTION

FUNCTION "ExtractStringFromCharArray" : Word   // FC2, SCL
{ S7_Optimized_Access := 'TRUE' }
   VAR_INPUT
      textBefore : String;
      textAfter : String;
   END_VAR
   VAR_OUTPUT
      extractedString : String;
      status : Word;
   END_VAR
   VAR_IN_OUT
      searchIn : Variant;
   END_VAR
   VAR_TEMP
      tempNumElements : UDInt;
      tempPosInArray : DInt;
      tempLenTextBefore : Int;
      tempPosTextBefore : DInt;
      tempLenTextAfter : Int;
      tempPosTextAfter : Int;
      tempString : String;
   END_VAR
   VAR CONSTANT
      LEN_STRING : UInt := 254;
      STATUS_TEXT_FOUND : Word := 16#0000;
      WARNING_ONLY_START : Word := 16#9001;
      WARNING_NOTHING_FOUND : Word := 16#9002;
      STATUS_NO_ERROR : Word := 16#0000;
      ERR_NO_ARRAY : Word := 16#8200;
   END_VAR
BEGIN
   REGION BLOCK INFO HEADER
       //===============================================================================
       // Title:            ExtractStringFromCharArray
       // Function:         The function extracts a String specified by a text before and after
       //                   from an array of characters.

       //===============================================================================
   END_REGION

   REGION Initialization
       #tempPosTextBefore := 0;
       #tempPosTextAfter := 0;
       #tempPosInArray := 0;
       #tempLenTextBefore := LEN(#textBefore);
       #tempLenTextAfter := LEN(#textAfter);
       #extractedString := '';
       #status := #STATUS_NO_ERROR;
       #ExtractStringFromCharArray := #WARNING_NOTHING_FOUND;

       REGION Validation of inputs
           // check whether the input is an ARRAY and TYPE of elements is CHAR or BYTE
           // IF so, the number OF the ARRAY elements is read out.
           // IF it is NOT an ARRAY, the program execution is terminated at this point
           IF TRUE
               AND IS_ARRAY(#searchIn)
               AND ((TypeOfElements(#searchIn) = Char) OR (TypeOfElements(#searchIn) = Byte))
           THEN
               // Get number of elements
               #tempNumElements := CountOfElements(#searchIn);
           ELSE
               #status := #ERR_NO_ARRAY;
               RETURN;
           END_IF;
       END_REGION Validation of inputs
   END_REGION Initialization

   REGION Process
       REPEAT // Search for text before until something was found
           // Convert Chars to String
           Chars_TO_Strg(Chars := #searchIn,
                         pChars := #tempPosInArray, // Subtract offset since pChars is zero based
                         Cnt := UDINT_TO_UINT(MIN(IN1 := #LEN_STRING, IN2 := #tempNumElements)),
                         Strg => #tempString);

           // Search for text before
           #tempPosTextBefore := FIND(IN1 := #tempString, IN2 := #textBefore);

           // Text before was found
           IF #tempPosTextBefore > 0 THEN
               // Set position in array to end of text before
               #tempPosInArray += #tempPosTextBefore + #tempLenTextBefore - 1;

               // Create new string from end of text before
               Chars_TO_Strg(Chars := #searchIn,
                             pChars := #tempPosInArray, // Subtract offset since pChars is zero based
                             Cnt := UDINT_TO_UINT(MIN(IN1 := #LEN_STRING, IN2 := #tempNumElements)),
                             Strg => #tempString);

               // Find end of string to be extracted
               #tempPosTextAfter := FIND(IN1 := #tempString, IN2 := #textAfter);

               IF #tempPosTextAfter > 0 THEN // Shorten string if text after was found
                   #extractedString := LEFT(IN := #tempString, L := #tempPosTextAfter - 1);
                   #ExtractStringFromCharArray := #STATUS_TEXT_FOUND;
                   EXIT;

               ELSE // Output whole string if text after was not found
                   #extractedString := #tempString;
                   #ExtractStringFromCharArray := #WARNING_ONLY_START;
                   EXIT;
               END_IF;

           ELSE
               // Otherwise continue search in next string minus length of text before to ensure
               // keywords are not broken up at the end of a string and thus missed
               #tempPosInArray += UINT_TO_INT(#LEN_STRING) - #tempLenTextBefore;
           END_IF;

           // Repeat until end of array is reached
       UNTIL (#tempPosInArray > #tempNumElements) END_REPEAT;
   END_REGION Process
END_FUNCTION

FUNCTION "MatrixAddition" : Void   // FC3, SCL
{ S7_Optimized_Access := 'TRUE' }
   VAR_INPUT
      matrix1 : Array[*, *] of LReal;
      matrix2 : Array[*, *] of LReal;
   END_VAR
   VAR_OUTPUT
      error : Bool;
      status : Word;
   END_VAR
   VAR_IN_OUT
      matrixResult : Array[*, *] of LReal;
   END_VAR
   VAR_TEMP
      tempMatrix1LowerBoundRows : DInt;
      tempMatrix1LowerBoundColumns : DInt;
      tempMatrix1UpperBoundRows : DInt;
      tempMatrix1UpperBoundColumns : DInt;
      tempMatrix2LowerBoundRows : DInt;
      tempMatrix2LowerBoundColumns : DInt;
      tempMatrix2UpperBoundRows : DInt;
      tempMatrix2UpperBoundColumns : DInt;
      tempResultMatrixLowerBoundRows : DInt;
      tempResultMatrixLowerBoundColumns : DInt;
      tempResultMatrixUpperBoundRows : DInt;
      tempResultMatrixUpperBoundColumns : DInt;
      tempCounterRows : DInt;
      tempCounterColumns : DInt;
   END_VAR
   VAR CONSTANT
      ROWS : UInt := 1;
      COLUMNS : UInt := 2;
      STATUS_NO_ERROR : Word := 16#0000;
      ERR_MATR1_LOWBOUND_ROWS_MATR2_LOWBOUND_ROWS : Word := 16#8200;
      ERR_MATR1_LOWBOUND_ROWS_RESMATR_LOWBOUND_ROWS : Word := 16#8201;
      ERR_MATR1_LOWBOUND_COLUMNS_MATR2_LOWBOUND_COLUMNS : Word := 16#8202;
      ERR_MATR1_LOWBOUND_COLUMNS_RESMATR_LOWBOUND_COLUMNS : Word := 16#8203;
      ERR_MATR1_UPPBOUND_ROWS_MATR2_UPPBOUND_ROWS : Word := 16#8204;
      ERR_MATR1_UPPBOUND_ROWS_RESMATR_UPPBOUND_ROWS : Word := 16#8205;
      ERR_MATR1_UPPBOUND_COLUMNS_MATR2_UPPBOUND_COLUMNS : Word := 16#8206;
      ERR_MATR1_UPPBOUND_COLUMNS_RESMATR_UPPBOUND_COLUMNS : Word := 16#8207;
   END_VAR
BEGIN
   REGION Block info header
       //=============================================================================
       // Title:            MatrixAddition
       // Comment/Function: Caluclates the sum of two matrices

       //=============================================================================
   END_REGION Block info header

   REGION Getting matrices size
       //Determine the size of the matrices
       // Lower bound rows
       #tempMatrix1LowerBoundRows := LOWER_BOUND(ARR := #matrix1, DIM := #ROWS);
       #tempMatrix2LowerBoundRows := LOWER_BOUND(ARR := #matrix2, DIM := #ROWS);
       #tempResultMatrixLowerBoundRows := LOWER_BOUND(ARR := #matrixResult, DIM := #ROWS);
       // Lower bound columns
       #tempMatrix1LowerBoundColumns := LOWER_BOUND(ARR := #matrix1, DIM := #COLUMNS);
       #tempMatrix2LowerBoundColumns := LOWER_BOUND(ARR := #matrix2, DIM := #COLUMNS);
       #tempResultMatrixLowerBoundColumns := LOWER_BOUND(ARR := #matrixResult, DIM := #COLUMNS);

       // Upper bound rows
       #tempMatrix1UpperBoundRows := UPPER_BOUND(ARR := #matrix1, DIM := #ROWS);
       #tempMatrix2UpperBoundRows := UPPER_BOUND(ARR := #matrix2, DIM := #ROWS);
       #tempResultMatrixUpperBoundRows := UPPER_BOUND(ARR := #matrixResult, DIM := #ROWS);
       // Upper bound columns
       #tempMatrix1UpperBoundColumns := UPPER_BOUND(ARR := #matrix1, DIM := #COLUMNS);
       #tempMatrix2UpperBoundColumns := UPPER_BOUND(ARR := #matrix2, DIM := #COLUMNS);
       #tempResultMatrixUpperBoundColumns := UPPER_BOUND(ARR := #matrixResult, DIM := #COLUMNS);
   END_REGION

   REGION Error evaluation of matrixes dimentions
       //Check the lower bound of all matrices
       IF (#tempMatrix1LowerBoundRows <> #tempMatrix2LowerBoundRows) THEN
           #error := TRUE;
           #status := #ERR_MATR1_LOWBOUND_ROWS_MATR2_LOWBOUND_ROWS;
           RETURN;
       ELSIF (#tempMatrix1LowerBoundRows <> #tempResultMatrixLowerBoundRows) THEN
           #error := TRUE;
           #status := #ERR_MATR1_LOWBOUND_ROWS_RESMATR_LOWBOUND_ROWS;
           RETURN;
       ELSIF (#tempMatrix1LowerBoundColumns <> #tempMatrix2LowerBoundColumns) THEN
           #error := TRUE;
           #status := #ERR_MATR1_LOWBOUND_COLUMNS_MATR2_LOWBOUND_COLUMNS;
           RETURN;
       ELSIF (#tempMatrix1LowerBoundColumns <> #tempResultMatrixLowerBoundColumns) THEN
           #error := TRUE;
           #status := #ERR_MATR1_LOWBOUND_COLUMNS_RESMATR_LOWBOUND_COLUMNS;
           RETURN;
       END_IF;
       //Check the upper bound of all matrices
       IF (#tempMatrix1UpperBoundRows <> #tempMatrix2UpperBoundRows) THEN
           #error := TRUE;
           #status := #ERR_MATR1_UPPBOUND_ROWS_MATR2_UPPBOUND_ROWS;
           RETURN;
       ELSIF (#tempMatrix1UpperBoundRows <> #tempResultMatrixUpperBoundRows) THEN
           #error := TRUE;
           #status := #ERR_MATR1_UPPBOUND_ROWS_RESMATR_UPPBOUND_ROWS;
           RETURN;
       ELSIF (#tempMatrix1UpperBoundColumns <> #tempMatrix2UpperBoundColumns) THEN
           #error := TRUE;
           #status := #ERR_MATR1_UPPBOUND_COLUMNS_MATR2_UPPBOUND_COLUMNS;
           RETURN;
       ELSIF (#tempMatrix1UpperBoundColumns <> #tempResultMatrixUpperBoundColumns) THEN
           #error := TRUE;
           #status := #ERR_MATR1_UPPBOUND_COLUMNS_RESMATR_UPPBOUND_COLUMNS;
           RETURN;
       END_IF;
   END_REGION

   REGION Addition of the matrices and writting to output
       FOR #tempCounterRows := #tempMatrix1LowerBoundRows TO #tempMatrix1UpperBoundRows DO
           FOR #tempCounterColumns := #tempMatrix1LowerBoundColumns TO #tempMatrix1UpperBoundColumns DO
               #matrixResult[#tempCounterRows, #tempCounterColumns] := #matrix1[#tempCounterRows, #tempCounterColumns] + #matrix2[#tempCounterRows, #tempCounterColumns];
           END_FOR;
       END_FOR;

       #error := false;
       #status := #STATUS_NO_ERROR;
       // ENO mechanism is not used
       ENO := TRUE;
   END_REGION
END_FUNCTION

FUNCTION "RandomRange_DInt" : DInt   // FC5, SCL
{ S7_Optimized_Access := 'TRUE' }
   VAR_INPUT
      minValue : DInt;
      maxValue : DInt;
   END_VAR
   VAR_OUTPUT
      error : Bool;
      status : Word;
   END_VAR
   VAR_TEMP
      tempTime : DTL;
      tempNanoSecondInDWord : DWord;
      tempTimeStatus : Word;
      tempRandomValue : DWord;
      tempNormReal : Real;
   END_VAR
   VAR CONSTANT
      ZERO : DInt := 0;
      MAX_UDINT : UDInt := 4_294_967_295;
      SUB_STATUS_NO_ERROR : Word := 16#0000;
      STATUS_FINISHED_NO_ERROR : Word := 16#0000;
      ERR_MAX_LESS_MIN : Word := 16#8200;
      ERR_RD_SYS_T : Word := 16#8600;
   END_VAR
BEGIN
   REGION Block info header
       //=============================================================================
       // Title:            RandomRange_DInt
       // Comment/Function: This function generates random numbers in defined limits (Datatype DInt)

       //=============================================================================
   END_REGION Block info header

   REGION Validation
       // Check if the maximal Value is less than the minimal value
       IF (#minValue > #maxValue) THEN
           #error := true;
           #status := #ERR_MAX_LESS_MIN;

           #RandomRange_DInt := #ZERO;
           RETURN;
       END_IF;

       // Read system time
       #tempTimeStatus := INT_TO_WORD(RD_SYS_T(#tempTime));

       // Check return variable for error
       IF (#tempTimeStatus <> #SUB_STATUS_NO_ERROR) THEN
           #error := true;
           #status := #ERR_RD_SYS_T;

           #RandomRange_DInt := #ZERO;
           RETURN;
       END_IF;
   END_REGION

   REGION Calculating random number
       // Converting to double word so individual bytes can be addressed
       #tempNanoSecondInDWord := UDINT_TO_DWORD(#tempTime.NANOSECOND);

       // Callculate a random-start-value depending on the time
       #tempRandomValue.%B3 := #tempNanoSecondInDWord.%B0;
       #tempRandomValue.%B2 := #tempNanoSecondInDWord.%B1;
       #tempRandomValue.%B1 := #tempNanoSecondInDWord.%B2;
       #tempRandomValue.%B0 := #tempNanoSecondInDWord.%B3;

       // Norm the calculated random number: 0.0 <= #tempNormReal <= 1.0
       #tempNormReal := UDINT_TO_REAL(DWORD_TO_UDINT(#tempRandomValue)) / UDINT_TO_REAL(#MAX_UDINT);

       // Scale the tempNormReal to be in the range of maxValue and minValue
       #RandomRange_DInt := REAL_TO_DINT((#tempNormReal * DINT_TO_REAL(#maxValue - #minValue) + DINT_TO_REAL(#minValue)));

       #error := false;
       #status := #STATUS_FINISHED_NO_ERROR;

       // ENO mechanism is not used
       ENO := TRUE;
   END_REGION
END_FUNCTION

FUNCTION "SearchMinMax_DInt" : Void   // FC6, SCL
{ S7_Optimized_Access := 'TRUE' }
   VAR_INPUT
      values : Array[*] of DInt;
   END_VAR
   VAR_OUTPUT
      minValue : DInt;
      minValueIndex : DInt;
      maxValue : DInt;
      maxValueIndex : DInt;
   END_VAR
   VAR_TEMP
      tempArrayLowerBound : DInt;
      tempArrayUpperBound : DInt;
      tempCounter : DInt;
      tempArrayIndexMax : DInt;
      tempArrayIndexMin : DInt;
      tempActValue : DInt;
      tempMinValue : DInt;
      tempMaxValue : DInt;
   END_VAR
   VAR CONSTANT
      START_FROM_SECOND_ELEMENT : Int := 1;
      DIMENSION_ONE : UInt := 1;
   END_VAR
BEGIN
   REGION Block info header
       //=============================================================================
       // Title:            SearchMinMax_DInt
       // Comment/Function: Searches an array for the minimum and maximum number and
       //                   outputs the position and values of those numbers for
       //                   array of double integers

       //=============================================================================
   END_REGION Block info header

   REGION Validation of inputs and outputs 
       // Lower bound
       #tempArrayLowerBound := LOWER_BOUND(ARR := #values, DIM := #DIMENSION_ONE);
       // Upper bound 
       #tempArrayUpperBound := UPPER_BOUND(ARR := #values, DIM := #DIMENSION_ONE);
   END_REGION

   REGION Searching the array 
       // Assign first value as min / max
       #tempMinValue := #tempMaxValue := #values[#tempArrayLowerBound];
       #tempArrayIndexMin := #tempArrayIndexMax := #tempArrayLowerBound;

       // Search the Array for min/max values
       FOR #tempCounter := (#tempArrayLowerBound + #START_FROM_SECOND_ELEMENT) TO #tempArrayUpperBound DO

           #tempActValue := #values[#tempCounter];

           // check for min
           IF #tempActValue < #tempMinValue THEN
               #tempMinValue := #tempActValue;
               #tempArrayIndexMin := #tempCounter;
               // check for max
           ELSIF #tempActValue > #tempMaxValue THEN
               #tempMaxValue := #tempActValue;
               #tempArrayIndexMax := #tempCounter;
           END_IF;
       END_FOR;
   END_REGION

   REGION Writting to outputs
       // Copy found values to outputs
       // Copy Minimum value
       #minValue := #values[#tempArrayIndexMin];
       // Copy Maximum value
       #maxValue := #values[#tempArrayIndexMax];

       // Write found indexes to outputs
       #minValueIndex := #tempArrayIndexMin;
       #maxValueIndex := #tempArrayIndexMax;

       // ENO mechanism is not used, no error possible
       ENO := TRUE;
   END_REGION
END_FUNCTION

FUNCTION "StringToTaddr" : TADDR_Param   // FC7, SCL
{ S7_Optimized_Access := 'TRUE' }
   VAR_INPUT
      ipAddressString : String;
   END_VAR
   VAR_OUTPUT
      error : Bool;
      status : Word;
   END_VAR
   VAR_TEMP
      tempOctetIndex : Int;
      tempCharPosition : Int;
      tempAddressString : String;
      tempOctetString : String[#MAX_CHAR_FOR_IP_OCTET_NUMBER];
      tempNumber : UDInt;
      tempPortNumberIsSpecified : Bool;
      tempIpAdressTaddr : TADDR_Param;
   END_VAR
   VAR CONSTANT
      STATUS_FINISHED_NO_ERROR : Word := 16#0000;
      ERR_OCTET_WRONG_NUMBER_OF_CHAR : Word := 16#8110;
      ERR_OCTET_STRING_IS_EMPTY : Word := 16#8120;
      ERR_OCTET_EXCEEDS_MAX_IP_ADDRESS : Word := 16#8130;
      ERR_PORT_WRONG_NUMBER_OF_CHAR : Word := 16#8150;
      ERR_PORT_STRING_IS_EMPTY : Word := 16#8151;
      ERR_PORT_EXCEEDS_MAX_PORT : Word := 16#8152;
      MAX_IP_ADDRESS_OCTET_NUMBER : USInt := 255;
      MAX_PORT_NUMBER : UInt := 65535;
      EMPTY_STRING : Int := 0;
      MAX_CHAR_FOR_IP_OCTET_NUMBER : Int := 4;
      MAX_CHAR_FOR_PORT_NUMBER : Int := 5;
      INIT_VAL : USInt := 0;
      NUMBER_OF_IP_OCTETS : Int := 4;
      CHAR_DOT : Char := '.';
      CHAR_COLON : Char := ':';
      CONVERT_FORMAT_TO_INTEGER : Word := 16#0000;
      CONVERT_START_POSITION : UInt := 1;
   END_VAR
BEGIN
   REGION BLOCK INFO HEADER
       //===============================================================================
       // Title:            StringToTaddr
       // Comment/Function: This function converts a string IP Address into TADDR Parameter format.

       //=============================================================================
   END_REGION Block info header

   REGION Initialization
       #tempAddressString := #ipAddressString;
       #tempIpAdressTaddr.REM_IP_ADDR[1] := #INIT_VAL;
       #tempIpAdressTaddr.REM_IP_ADDR[2] := #INIT_VAL;
       #tempIpAdressTaddr.REM_IP_ADDR[3] := #INIT_VAL;
       #tempIpAdressTaddr.REM_IP_ADDR[4] := #INIT_VAL;
       #tempIpAdressTaddr.REM_PORT_NR := #INIT_VAL;
       #StringToTaddr := #tempIpAdressTaddr;
   END_REGION

   REGION Process Address String  
       REGION Process octests 1-4
           FOR #tempOctetIndex := 1 TO #NUMBER_OF_IP_OCTETS BY 1 DO
               // check if loop has not reached the last octet
               IF #tempOctetIndex < #NUMBER_OF_IP_OCTETS THEN
                   // search for dot as octet seperator
                   // there has to be a dot present between the octets
                   #tempCharPosition := FIND(IN1 := #tempAddressString, IN2 := #CHAR_DOT);

               ELSE
                   // search for colon as port seperator after the last Octet
                   #tempCharPosition := FIND(IN1 := #tempAddressString, IN2 := #CHAR_COLON);

                   // if colon is present, there is a port number specified / check if Port number added
                   #tempPortNumberIsSpecified := (#tempCharPosition > 0);

                   // if no port is spezified, its just the last octet
                   IF NOT #tempPortNumberIsSpecified THEN
                       // need to set the char position to the end of string + one for later cobesion and checks
                       #tempCharPosition := LEN(#tempAddressString) + 1;
                   END_IF;
               END_IF;

               REGION Octet conversion
                   // check if IP Octet contains more then three digits --> Error
                   IF #tempCharPosition > #MAX_CHAR_FOR_IP_OCTET_NUMBER THEN
                       #error := TRUE;
                       #status := #ERR_OCTET_WRONG_NUMBER_OF_CHAR OR INT_TO_WORD(#tempOctetIndex);
                       #StringToTaddr := #tempIpAdressTaddr;
                       RETURN;
                   END_IF;

                   // extract octet string
                   #tempOctetString := LEFT(IN := #tempAddressString, L := #tempCharPosition - 1);
                   // Check if Octet string is empty --> Error
                   IF LEN(#tempOctetString) = #EMPTY_STRING THEN
                       #error := TRUE;
                       #status := #ERR_OCTET_STRING_IS_EMPTY OR INT_TO_WORD(#tempOctetIndex);
                       #StringToTaddr := #tempIpAdressTaddr;
                       RETURN;
                   END_IF;

                   // Convert the octet string to numerical value
                   STRG_VAL(IN := #tempOctetString,
                            FORMAT := #CONVERT_FORMAT_TO_INTEGER,
                            P := #CONVERT_START_POSITION,
                            OUT => #tempNumber);

                   // check if the octet number exeeds the maximum possible range of 255 of USInt --> Error
                   IF #tempNumber > #MAX_IP_ADDRESS_OCTET_NUMBER THEN
                       #error := TRUE;
                       #status := #ERR_OCTET_EXCEEDS_MAX_IP_ADDRESS OR INT_TO_WORD(#tempOctetIndex);
                       #StringToTaddr := #tempIpAdressTaddr;
                       RETURN;
                   END_IF;

                   // add address octet to temp address tag
                   #tempIpAdressTaddr.REM_IP_ADDR[#tempOctetIndex] := UDINT_TO_USINT(#tempNumber);

                   // delete octet string from address string
                   #tempAddressString := DELETE(IN := #tempAddressString, P := 1, L := #tempCharPosition);
               END_REGION Octet conversion
           END_FOR;
       END_REGION Process octests 1-4

       REGION PORT number conversion
           // If the string contains a port number too, parse it
           IF #tempPortNumberIsSpecified THEN
               // lenght of string exceeds length of port string --> Error
               IF LEN(#tempAddressString) > #MAX_CHAR_FOR_PORT_NUMBER THEN
                   #error := TRUE;
                   #status := #ERR_PORT_WRONG_NUMBER_OF_CHAR;
                   #StringToTaddr := #tempIpAdressTaddr;
                   RETURN;

                   // Check if string is empty --> Error
               ELSIF LEN(#tempAddressString) = #EMPTY_STRING THEN
                   #error := TRUE;
                   #status := #ERR_PORT_STRING_IS_EMPTY;
                   #StringToTaddr := #tempIpAdressTaddr;
                   RETURN;
               END_IF;

               // Convert the port number string to numerical value
               STRG_VAL(IN := #tempAddressString,
                        FORMAT := #CONVERT_FORMAT_TO_INTEGER,
                        P := #CONVERT_START_POSITION,
                        OUT => #tempNumber);

               // check if the Port number exeeds the maximum possible range of 65535 of UInt --> Error
               IF #tempNumber > #MAX_PORT_NUMBER THEN
                   #error := TRUE;
                   #status := #ERR_PORT_EXCEEDS_MAX_PORT;
                   #StringToTaddr := #tempIpAdressTaddr;
                   RETURN;
               END_IF;

               // add port number to temp address tag
               #tempIpAdressTaddr.REM_PORT_NR := UDINT_TO_UINT(#tempNumber);
           END_IF;
       END_REGION PORT number conversion

   END_REGION

   REGION Outputs
       #error := FALSE;
       #status := #STATUS_FINISHED_NO_ERROR;
       #StringToTaddr := #tempIpAdressTaddr;
       //ENO mechanism is not used - forced to true.
       ENO := TRUE;
   END_REGION
END_FUNCTION

FUNCTION "MatrixAux" : Void   // FC8, SCL
{ S7_Optimized_Access := 'TRUE' }
VERSION : 0.1
   VAR_TEMP
      count : Int;
   END_VAR
BEGIN
   FOR #count := 1 TO 2 DO

       "MatrixAddition_DB".matrix1[1,#count]:="MatrixAddition_DBG".matrix1[#count];
   END_FOR;

   FOR #count := 1 TO 2 DO

       "MatrixAddition_DB".matrix1[2, #count] := "MatrixAddition_DBG".matrix1[#count + 2];
   END_FOR;

   FOR #count := 1 TO 2 DO

       "MatrixAddition_DB".matrix2[1, #count] := "MatrixAddition_DBG".matrix2[#count];
   END_FOR;

   FOR #count := 1 TO 2 DO

       "MatrixAddition_DB".matrix2[2, #count] := "MatrixAddition_DBG".matrix2[#count + 2];
   END_FOR;

   FOR #count := 1 TO 2 DO

       "MatrixAddition_DBG".matrixResult[#count] := "MatrixAddition_DB".matrixResult[1, #count];
   END_FOR;

   FOR #count := 1 TO 2 DO

       "MatrixAddition_DBG".matrixResult[#count + 2] := "MatrixAddition_DB".matrixResult[2, #count];
   END_FOR;
END_FUNCTION

FUNCTION "MatrixAux_1" : Void   // FC9, SCL
{ S7_Optimized_Access := 'TRUE' }
VERSION : 0.1
   VAR_TEMP
      count : Int;
   END_VAR
BEGIN
   FOR #count := 1 TO 2 DO

       "MatrixAddition_DB".matrix1[1,#count]:="MatrixAddition_DBG".matrix1[#count];
   END_FOR;

   FOR #count := 1 TO 2 DO

       "MatrixAddition_DB".matrix1[2, #count] := "MatrixAddition_DBG".matrix1[#count + 2];
   END_FOR;

   FOR #count := 1 TO 2 DO

       "MatrixAddition_DB".matrix2[1, #count] := "MatrixAddition_DBG".matrix2[#count];
   END_FOR;

   FOR #count := 1 TO 2 DO

       "MatrixAddition_DB".matrix2[2, #count] := "MatrixAddition_DBG".matrix2[#count + 2];
   END_FOR;

   FOR #count := 1 TO 2 DO

       "MatrixAddition_DBG".matrixResult[#count] := "MatrixAddition_DB".matrixResult[1, #count];
   END_FOR;

   FOR #count := 1 TO 2 DO

       "MatrixAddition_DBG".matrixResult[#count + 2] := "MatrixAddition_DB".matrixResult[2, #count];
   END_FOR;
END_FUNCTION

ORGANIZATION_BLOCK "Main"   // OB1, LAD, ProgramCycle
TITLE = "Main Program Sweep (Cycle)"
{ S7_Optimized_Access := 'TRUE' }
VERSION : 0.1
   VAR_INPUT
      Initial_Call : Bool;   // Initial call of this OB
      Remanence : Bool;   // =True, if remanent data are available
   END_VAR
BEGIN

REGION Network 1
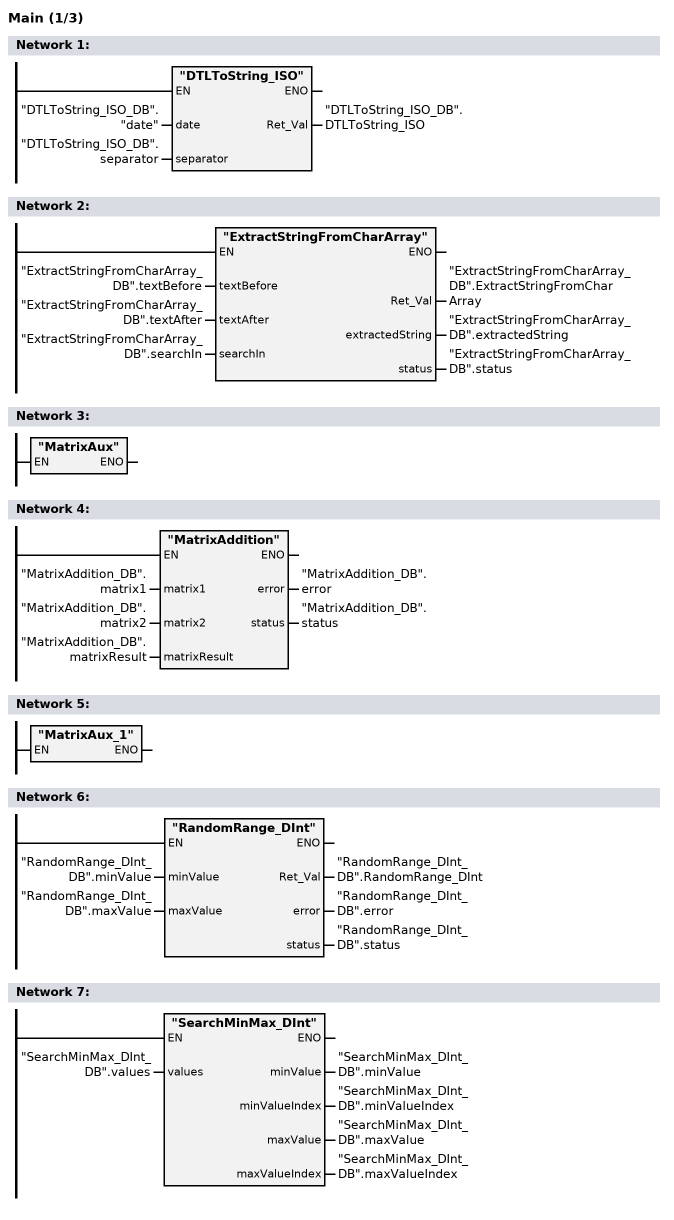
   RUNG wire#powerrail
      "DTLToString_ISO"("date" := "DTLToString_ISO_DB"."date", separator := "DTLToString_ISO_DB".separator, Ret_Val => "DTLToString_ISO_DB".DTLToString_ISO)
   END_RUNG
   // the same network as SCL:
   "DTLToString_ISO_DB".DTLToString_ISO := "DTLToString_ISO"("date" := "DTLToString_ISO_DB"."date",
                           separator := "DTLToString_ISO_DB".separator);
END_REGION

REGION Network 2
   RUNG wire#powerrail
      "ExtractStringFromCharArray"(textBefore := "ExtractStringFromCharArray_DB".textBefore, textAfter := "ExtractStringFromCharArray_DB".textAfter, searchIn := "ExtractStringFromCharArray_DB".searchIn, Ret_Val => "ExtractStringFromCharArray_DB".ExtractStringFromCharArray, extractedString => "ExtractStringFromCharArray_DB".extractedString, status => "ExtractStringFromCharArray_DB".status)
   END_RUNG
   // the same network as SCL:
   "ExtractStringFromCharArray_DB".ExtractStringFromCharArray := "ExtractStringFromCharArray"(textBefore := "ExtractStringFromCharArray_DB".textBefore,
                           textAfter := "ExtractStringFromCharArray_DB".textAfter,
                           searchIn := "ExtractStringFromCharArray_DB".searchIn,
                           extractedString => "ExtractStringFromCharArray_DB".extractedString,
                           status => "ExtractStringFromCharArray_DB".status);
END_REGION

REGION Network 3
   RUNG wire#powerrail
      "MatrixAux"()
   END_RUNG
   // the same network as SCL:
   "MatrixAux"();
END_REGION

REGION Network 4
   RUNG wire#powerrail
      "MatrixAddition"(matrix1 := "MatrixAddition_DB".matrix1, matrix2 := "MatrixAddition_DB".matrix2, matrixResult := "MatrixAddition_DB".matrixResult, error => "MatrixAddition_DB".error, status => "MatrixAddition_DB".status)
   END_RUNG
   // the same network as SCL:
   "MatrixAddition"(matrix1 := "MatrixAddition_DB".matrix1,
                    matrix2 := "MatrixAddition_DB".matrix2,
                    matrixResult := "MatrixAddition_DB".matrixResult,
                    error => "MatrixAddition_DB".error,
                    status => "MatrixAddition_DB".status);
END_REGION

REGION Network 5
   RUNG wire#powerrail
      "MatrixAux_1"()
   END_RUNG
   // the same network as SCL:
   "MatrixAux_1"();
END_REGION

REGION Network 6
   RUNG wire#powerrail
      "RandomRange_DInt"(minValue := "RandomRange_DInt_DB".minValue, maxValue := "RandomRange_DInt_DB".maxValue, Ret_Val => "RandomRange_DInt_DB".RandomRange_DInt, error => "RandomRange_DInt_DB".error, status => "RandomRange_DInt_DB".status)
   END_RUNG
   // the same network as SCL:
   "RandomRange_DInt_DB".RandomRange_DInt := "RandomRange_DInt"(minValue := "RandomRange_DInt_DB".minValue,
                           maxValue := "RandomRange_DInt_DB".maxValue,
                           error => "RandomRange_DInt_DB".error,
                           status => "RandomRange_DInt_DB".status);
END_REGION

REGION Network 7
   RUNG wire#powerrail
      "SearchMinMax_DInt"(values := "SearchMinMax_DInt_DB".values, minValue => "SearchMinMax_DInt_DB".minValue, minValueIndex => "SearchMinMax_DInt_DB".minValueIndex, maxValue => "SearchMinMax_DInt_DB".maxValue, maxValueIndex => "SearchMinMax_DInt_DB".maxValueIndex)
   END_RUNG
   // the same network as SCL:
   "SearchMinMax_DInt"(values := "SearchMinMax_DInt_DB".values,
                       minValue => "SearchMinMax_DInt_DB".minValue,
                       minValueIndex => "SearchMinMax_DInt_DB".minValueIndex,
                       maxValue => "SearchMinMax_DInt_DB".maxValue,
                       maxValueIndex => "SearchMinMax_DInt_DB".maxValueIndex);
END_REGION

REGION Network 8
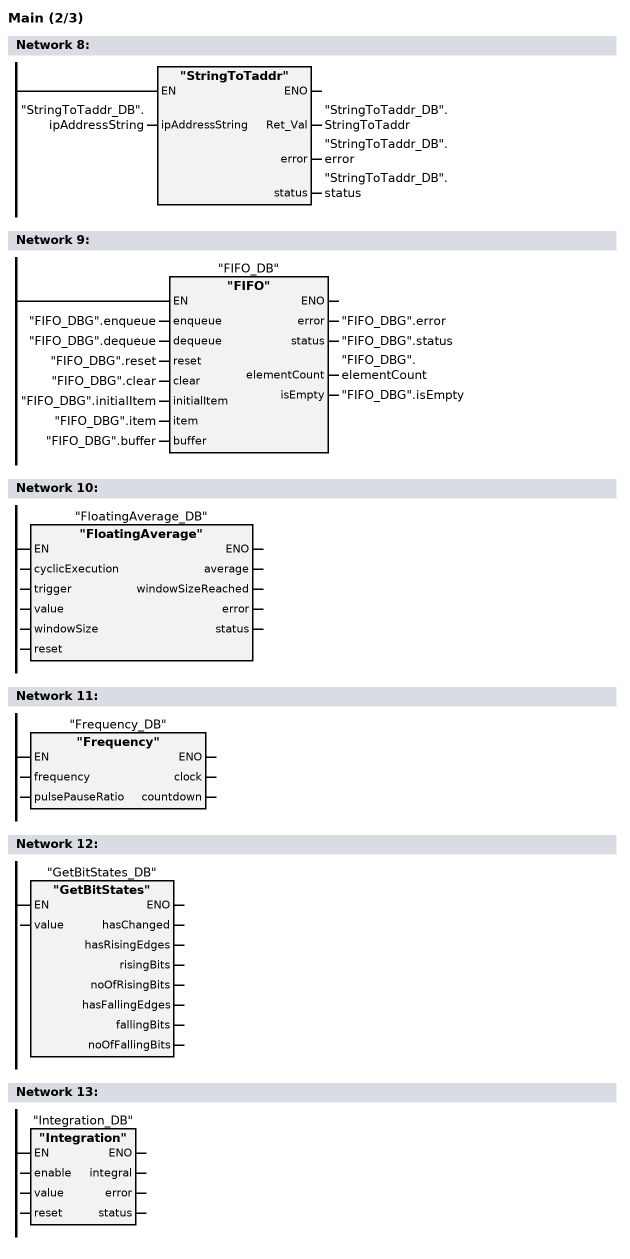
   RUNG wire#powerrail
      "StringToTaddr"(ipAddressString := "StringToTaddr_DB".ipAddressString, Ret_Val => "StringToTaddr_DB".StringToTaddr, error => "StringToTaddr_DB".error, status => "StringToTaddr_DB".status)
   END_RUNG
   // the same network as SCL:
   "StringToTaddr_DB".StringToTaddr := "StringToTaddr"(ipAddressString := "StringToTaddr_DB".ipAddressString,
                           error => "StringToTaddr_DB".error,
                           status => "StringToTaddr_DB".status);
END_REGION

REGION Network 9
   RUNG wire#powerrail
      "FIFO_DB"(enqueue := "FIFO_DBG".enqueue, dequeue := "FIFO_DBG".dequeue, reset := "FIFO_DBG".reset, clear := "FIFO_DBG".clear, initialItem := "FIFO_DBG".initialItem, item := "FIFO_DBG".item, buffer := "FIFO_DBG".buffer, error => "FIFO_DBG".error, status => "FIFO_DBG".status, elementCount => "FIFO_DBG".elementCount, isEmpty => "FIFO_DBG".isEmpty)
   END_RUNG
   // the same network as SCL:
   "FIFO_DB"(enqueue := "FIFO_DBG".enqueue,   // "FIFO"
             dequeue := "FIFO_DBG".dequeue,
             reset := "FIFO_DBG".reset,
             clear := "FIFO_DBG".clear,
             initialItem := "FIFO_DBG".initialItem,
             item := "FIFO_DBG".item,
             buffer := "FIFO_DBG".buffer,
             error => "FIFO_DBG".error,
             status => "FIFO_DBG".status,
             elementCount => "FIFO_DBG".elementCount,
             isEmpty => "FIFO_DBG".isEmpty);
END_REGION

REGION Network 10
   RUNG wire#powerrail
      "FloatingAverage_DB"(cyclicExecution :=, trigger :=, value :=, windowSize :=, reset :=, average =>, windowSizeReached =>, error =>, status =>)
   END_RUNG
   // the same network as SCL:
   "FloatingAverage_DB"();   // "FloatingAverage"
END_REGION

REGION Network 11
   RUNG wire#powerrail
      "Frequency_DB"(frequency :=, pulsePauseRatio :=, clock =>, countdown =>)
   END_RUNG
   // the same network as SCL:
   "Frequency_DB"();   // "Frequency"
END_REGION

REGION Network 12
   RUNG wire#powerrail
      "GetBitStates_DB"(value :=, hasChanged =>, hasRisingEdges =>, risingBits =>, noOfRisingBits =>, hasFallingEdges =>, fallingBits =>, noOfFallingBits =>)
   END_RUNG
   // the same network as SCL:
   "GetBitStates_DB"();   // "GetBitStates"
END_REGION

REGION Network 13
   RUNG wire#powerrail
      "Integration_DB"(enable :=, value :=, reset :=, integral =>, error =>, status =>)
   END_RUNG
   // the same network as SCL:
   "Integration_DB"();   // "Integration"
END_REGION

REGION Network 14
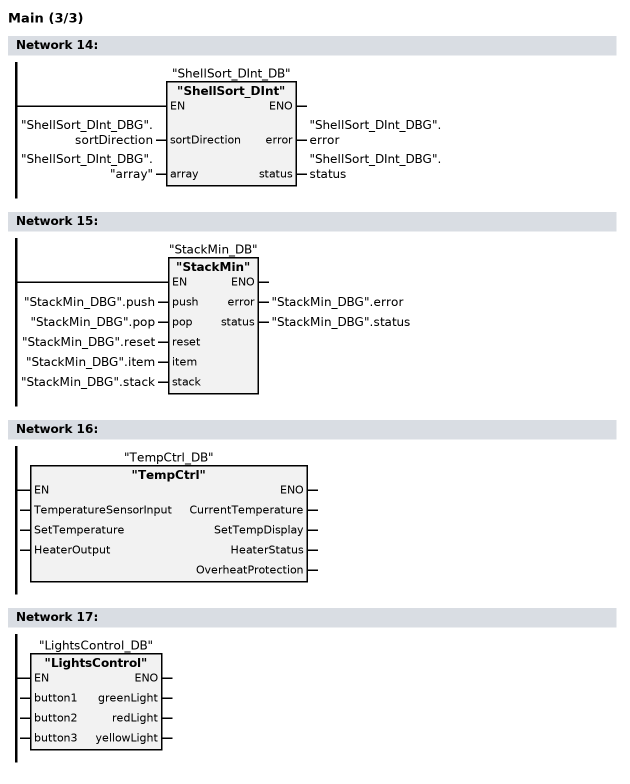
   RUNG wire#powerrail
      "ShellSort_DInt_DB"(sortDirection := "ShellSort_DInt_DBG".sortDirection, "array" := "ShellSort_DInt_DBG"."array", error => "ShellSort_DInt_DBG".error, status => "ShellSort_DInt_DBG".status)
   END_RUNG
   // the same network as SCL:
   "ShellSort_DInt_DB"(sortDirection := "ShellSort_DInt_DBG".sortDirection,   // "ShellSort_DInt"
                       "array" := "ShellSort_DInt_DBG"."array",
                       error => "ShellSort_DInt_DBG".error,
                       status => "ShellSort_DInt_DBG".status);
END_REGION

REGION Network 15
   RUNG wire#powerrail
      "StackMin_DB"(push := "StackMin_DBG".push, pop := "StackMin_DBG".pop, reset := "StackMin_DBG".reset, item := "StackMin_DBG".item, stack := "StackMin_DBG".stack, error => "StackMin_DBG".error, status => "StackMin_DBG".status)
   END_RUNG
   // the same network as SCL:
   "StackMin_DB"(push := "StackMin_DBG".push,   // "StackMin"
                 pop := "StackMin_DBG".pop,
                 reset := "StackMin_DBG".reset,
                 item := "StackMin_DBG".item,
                 stack := "StackMin_DBG".stack,
                 error => "StackMin_DBG".error,
                 status => "StackMin_DBG".status);
END_REGION

REGION Network 16
   RUNG wire#powerrail
      "TempCtrl_DB"(TemperatureSensorInput :=, SetTemperature :=, HeaterOutput :=, CurrentTemperature =>, SetTempDisplay =>, HeaterStatus =>, OverheatProtection =>)
   END_RUNG
   // the same network as SCL:
   "TempCtrl_DB"();   // "TempCtrl"
END_REGION

REGION Network 17
   RUNG wire#powerrail
      "LightsControl_DB"(button1 :=, button2 :=, button3 :=, greenLight =>, redLight =>, yellowLight =>)
   END_RUNG
   // the same network as SCL:
   "LightsControl_DB"();   // "LightsControl"
END_REGION
END_ORGANIZATION_BLOCK

// ===== library types =====

// folder: LGF/2 Counter operations

FUNCTION_BLOCK "LGF_GetBitStates"   // FB10018, SCL
TITLE = LGF_GetBitStates
{ S7_Optimized_Access := 'TRUE' }
AUTHOR : Siemens_Simatic_Systems_Support
FAMILY : LGF
NAME : LGF_CountBitStates
// This function checks a DWord for falling as well as rising edges.  
// It returns the number of edges, a DWord with the edge bits, and a boolean value if edge(s) are present.
// Diese Funktion prüft ein DWord auf fallende als auch steigende Flanken.  
// Sie liefert die Anzahl der Flanken, ein DWord mit den Flankenbits sowie eineb Boolschen Wert, falls Flanke(n) vorhanden sind.
   VAR_INPUT
      value : DWord;   // Check input value for changes and edges / Eingangswert auf Änderungen und Flanken prüfen
   END_VAR
   VAR_OUTPUT
      hasChanged : Bool;   // Input value has changed (compared to the previous cycle) / Eingangswert hat sich geändert (im Vergleich zum vorherigen Zyklus)
      hasRisingEdges : Bool;   // Input value has rising edges / Eingangswert hat steigende Flanken
      risingBits : DWord;   // Bitstream with the rising edges / Bitstream mit den steigenden Flanken
      noOfRisingBits : USInt;   // Number of rising edges in the input value / Anzahl der steigenden Flanken im Eingangswert
      hasFallingEdges : Bool;   // Input value has falling edges / Eingangswert hat fallende Flanken
      fallingBits : DWord;   // Bitstream with the falling edges / Bitstream mit den fallenden Flanken
      noOfFallingBits : USInt;   // Number of falling edges in the input value / Anzahl der fallenden Flanken im Eingangswert
   END_VAR
   VAR
      statPreviousValue : DWord;   // Static memory for input value from previous cycle / Statischer Speicher für Eingangswert aus vorherigem Zyklus
   END_VAR
   VAR_TEMP
      tempRisingResult : DWord;   // Temp tag for output value - rising edges Result / Temp-Tag für Ausgabewert - steigende Flanken Ergebnis
      tempNoRisingBits : DWord;   // Temp. tag for output value - number of rising bits Result / Temp-Tag für Ausgabewert - Anzahl der steigenden Bits Ergebnis
      tempFallingResult : DWord;   // Temp tag for output value - falling edges result / Temp-Tag für Ausgangswert - fallende Flanken Ergebnis
      tempNoFallingBits : DWord;   // Temp tag for output value - number of falling bits Result / Temp-Tag für Ausgabewert - Anzahl der fallenden Bits Ergebnis
   END_VAR
   VAR CONSTANT
      ZERO_EDGES : DWord;   // Zero edges detected / Nullflanken erkannt
   END_VAR
BEGIN
   REGION BLOCK INFO HEADER
     //============================================================================
     // SIEMENS AG / (c)Copyright 2018
     //----------------------------------------------------------------------------
     // Title:            LGF_GetBitStates
     // Comment/Function: Check DWord for edges, falling as well as rising.  
     //                   Returns the number of edges, DWords with edge bits and a bool if edge(s) exists.
     //                   https://graphics.stanford.edu/~seander/bithacks.html#CountBitsSetParallel
     // Library/Family:   LGF (Library General Functions)
     // Author:           Siemens Simatic Systems Support
     // Tested with:      1516F FW2.8 / S7-PLCSIM Advanced V3.0
     // Engineering:      TIA Portal V16 Update 4
     // Restrictions:     ENO not in use, set to true, no error handling
     // Requirements:     PLC (S7-1200 / S7-1500)
     //-------------------------------------------------------------------------------
     // Change log table:
     // Version  | Date       | Expert in charge        | Changes applied
     //----------|------------|-------------------------|------------------------------
     // 01.00.00 | 2021.01.28 | Simatic Systems Support | First released version
     //=============================================================================
   END_REGION BLOCK INFO HEADER

   REGION DESCRIPTION
   (/**/)
   END_REGION DESCRIPTION

   REGION PROGRAM LOGIC
     // Get edges from input DWord and DWord from previous cycle
     #tempRisingResult := #value AND NOT #statPreviousValue;
     #tempFallingResult := NOT #value AND #statPreviousValue;

     // Store value for next cycle
     #statPreviousValue := #value;

     // Copy edge result into work variable for counting the number of rising edges
     #tempNoRisingBits := #tempRisingResult;
     // Count number of rising edges, algorythm descriped from: https://graphics.stanford.edu/~seander/bithacks.html#CountBitsSetParallel
     #tempNoRisingBits := UDINT_TO_DWORD(DWORD_TO_UDINT(#tempNoRisingBits) - DWORD_TO_UDINT(SHR(IN := #tempNoRisingBits, N := 1) AND 16#55555555));
     #tempNoRisingBits := UDINT_TO_DWORD(DWORD_TO_UDINT(#tempNoRisingBits & 16#33333333) + DWORD_TO_UDINT(SHR(IN := #tempNoRisingBits, N := 2) AND 16#33333333));
     #tempNoRisingBits := SHR(IN := UDINT_TO_DWORD(DWORD_TO_UDINT(UDINT_TO_DWORD(DWORD_TO_UDINT(#tempNoRisingBits) + DWORD_TO_UDINT(SHR(IN := #tempNoRisingBits, N := 4))) AND 16#0F0F0F0F) * DWORD_TO_UDINT(16#01010101)), N := 24);

     // Copy edges result into work variable for counting the number of falling edges
     #tempNoFallingBits := #tempFallingResult;
     // Count number of falling edges, algorythm descriped from: https://graphics.stanford.edu/~seander/bithacks.html#CountBitsSetParallel
     #tempNoFallingBits := UDINT_TO_DWORD(DWORD_TO_UDINT(#tempNoFallingBits) - DWORD_TO_UDINT(SHR(IN := #tempNoFallingBits, N := 1) AND 16#55555555));
     #tempNoFallingBits := UDINT_TO_DWORD(DWORD_TO_UDINT(#tempNoFallingBits & 16#33333333) + DWORD_TO_UDINT(SHR(IN := #tempNoFallingBits, N := 2) AND 16#33333333));
     #tempNoFallingBits := SHR(IN := UDINT_TO_DWORD(DWORD_TO_UDINT(UDINT_TO_DWORD(DWORD_TO_UDINT(#tempNoFallingBits) + DWORD_TO_UDINT(SHR(IN := #tempNoFallingBits, N := 4))) AND 16#0F0F0F0F) * DWORD_TO_UDINT(16#01010101)), N := 24);
   END_REGION PROGRAM LOGIC

   REGION OUTPUTS
     #hasChanged := (#tempRisingResult > #ZERO_EDGES) OR (#tempFallingResult > #ZERO_EDGES);
     #hasRisingEdges := #tempRisingResult > #ZERO_EDGES;
     #risingBits := #tempRisingResult;
     #noOfRisingBits := DWORD_TO_USINT(#tempNoRisingBits);

     #hasFallingEdges := #tempFallingResult > #ZERO_EDGES;
     #fallingBits := #tempFallingResult;
     #noOfFallingBits := DWORD_TO_USINT(#tempNoFallingBits);

     // ENO not needed, no error evaluation needed
     ENO := FALSE;
   END_REGION OUTPUTS
END_FUNCTION_BLOCK

// folder: LGF/6 Converter operations

FUNCTION "LGF_DTLToString_ISO" : String   // FC10083, SCL
TITLE = LGF_DTLtoString_ISO
{ S7_Optimized_Access := 'TRUE' }
AUTHOR : Siemens_Digital_Industry
FAMILY : LGF
NAME : LGF_DTLtoString_ISO
// This function converts a date of data type DTL into a character string of data type STRING in international format (YYYY MM DD…). / Diese Funktion konvertiert ein Datum vom Datentyp DTL in eine Zeichenkette vom Datentyp STRING im internationalen Format (YYYY MM DD ...).
   VAR_INPUT
      "date" : DTL;   // Date to convert as DTL tag / Datum zum Konvertieren im Format DTL
      separator : Char;   // Separator between the components of the output date. / Trennzeichen zwischen den Komponenten des ausgegebenen Datums.
   END_VAR
   VAR_TEMP
      tempString : String;   // Temp string to setup the date string
      tempIndex : DInt;   // Temp iterator for replacing withspaces with '0' in nanosecondstring
   END_VAR
   // Ret_Val : Output string in accordance with the ISO 8601 format. Example: `2019-01-22 14:06:51.524621000`. / Ausgegebenen Zeichenkette entsprechend dem Format ISO 8601. Beispiel: `2019-01-22 14:06:51.524621000`.
   VAR CONSTANT
      CONVERT_SIZE_YEAR : USInt := 4;   // Number of character positions for Year
      CONVERT_SIZE_MONTH_DAY_HOUR_MINUTE_SECOND : USInt := 2;   // Number of character positions for Month, Day, Minute and Second
      CONVERT_SIZE_NANOSECOND : USInt := 9;   // Number of character positions for Nanoseconds
      CONVERT_PRECISION : USInt := 0;   // Number of decimal places to convert
      CONVERT_FORMAT_TO_STRING : Word := 16#0000;   // Output format of the characters
      CONVERT_START_POSITION_YEAR : UInt := 1;   // Character starting in string at which position the result is written.
      CONVERT_START_POSITION_MONTH : UInt := 6;   // Character starting in string at which position the result is written.
      CONVERT_START_POSITION_DAY : UInt := 9;   // Character starting in string at which position the result is written.
      CONVERT_START_POSITION_HOUR : UInt := 12;   // Character starting in string at which position the result is written.
      CONVERT_START_POSITION_MINUTE : UInt := 15;   // Character starting in string at which position the result is written.
      CONVERT_START_POSITION_SECOND : UInt := 18;   // Character starting in string at which position the result is written.
      CONVERT_START_POSITION_NANOSECOND : UInt := 21;   // Character starting in string at which position the result is written.
      SEPARATOR_POSITION_YEAR_MONTH : UInt := 5;   // Character starting in string at which position the result is written.
      SEPARATOR_POSITION_MONTH_DAY : UInt := 8;   // Character starting in string at which position the result is written.
      SEPARATOR_POSITION_HOUR_MINUTE : UInt := 14;   // Character starting in string at which position the result is written.
      SEPARATOR_POSITION_MINUTE_SECOND : UInt := 17;   // Character starting in string at which position the result is written.
      SEPARATOR_POSITION_SECOND_NANOSECOND : UInt := 20;   // Character starting in string at which position the result is written.
      SEPARATOR_NANOSECOND : Char := '.';   // Seperator for Nanosecond
      SEPARATOR_TIME : Char := ':';   // Seperator for Time
      SEPARATOR_DATE : Char := '-';   // Default separator for Date
      REPLACE_NANOSECOND_COUNT : DInt := 8;   // Number of Nonosecond characters to be checked for replacing withspaces wit '0'
   END_VAR
BEGIN
   REGION BLOCK INFO HEADER
     //===============================================================================
     // SIEMENS AG / (c)Copyright 2019
     //-------------------------------------------------------------------------------
     // Title:            LGF_DTLtoString_ISO
     // Comment/Function: This function converts a date of data type DTL into a character string of data type STRING in international format (YYYY MM DD…).
     // Library/Family:   LGF (Library General Functions)
     // Author:           Siemens Digital Industry Support
     // Tested with:      S7-PLCSIM Advanced V2.0 SP1
     // Engineering:      TIA Portal V15.1
     // Restrictions:     ENO mechanism is not used, no error handling
     // Requirements:     PLC (S7-1200 / S7-1500)
     //-------------------------------------------------------------------------------
     // Change log table:
     // Version  | Date       | Expert in charge       | Changes applied
     //----------|------------|------------------------|------------------------------
     // 01.00.00 | 15.06.2016 | Siemens Industry Online Support
     //                         First released version
     // 01.00.01 | 02.01.2017 | Siemens Industry Online Support
     //                         Upgrade: TIA Portal V14 Update 1
     // 01.00.02 | 17.08.2018 | Siemens Industry Online Support
     //                         Upgrade: TIA V15 Update 2
     // 01.00.03 | 23.11.2018 | Siemens Industry Online Support
     //                         Upgrade: TIA V15.1
     // 01.00.04 | 17.07.2019 | Simatic Systems Support
     //                         Bugfix - nanosecond precision and '0' filling
     // 01.00.05 | 18.07.2019 | Simatic Systems Support
     //                         Renamed from "LGF_DTLtoString" to "LGF_DTLtoString_ISO"
     //                         Split into two blocks, removed "format" input
     // 03.00.00 | 23.04.2020 | Simatic Systems Support | Set version to V3.0.0
     //                         Harmonize the version of the whole library
     // 03.00.01 | 23.02.2021 | Simatic Systems Support
     //                         Insert documentation
     //=============================================================================
   END_REGION Block info header

   REGION DESCRIPTION
     (/*The block reads a date of data type DTL and converts the individual components of the date (year, month, day, hour…) into a character string and outputs it in international format. The separator between the components of the date is variable.

   ##### International format (ISO 8601):

   {.imagePageWidth}
   ![LGF_DTLtoString_ISO - Structure of the character string in accordance with ISO 8601](LGF_DTLtoString_ISO.png "LGF_DTLtoString_ISO - Structure of the character string in accordance with ISO 8601")

   ##### Separator:

   At the input parameter `separatorDate`, you specify the separator between the components of the calendar date.

   ##### Example:

   * separatorDate = `/` - outString = `2016/03/16…`
   * separatorDate = `-` - outString = `2016-03-16…`
   Der Baustein liest ein Datum vom Datentyp DTL ein und konvertiert die einzelnen Komponenten des Datums (Jahr, Monat, Tag, Stunde...) in eine Zeichenkette und gibt diese im internationalen Format aus. Das Trennzeichen zwischen den Komponenten des Datums ist variabel.

   ##### Internationales Format (ISO 8601):

   {.imagePageWidth}
   ![LGF_DTLtoString_ISO - Aufbau der Zeichenkette nach ISO 8601](LGF_DTLtoString_ISO.png "LGF_DTLtoString_ISO - Aufbau der Zeichenkette nach ISO 8601")

   ##### Trennzeichen:

   Am Eingangsparameter `separatorDate` geben Sie das Trennzeichen zwischen den Komponenten des Kalenderdatums vor.

   ##### Beispiel:

   * separatorDate = `/` - outString = `2016/03/16…`
   * separatorDate = `-` - outString = `2016-03-16…`*/)
   END_REGION DESCRIPTION

   REGION INITIALISATION
     #tempString := '';
   END_REGION

   REGION CONVERTER
     // Set format parameters for output string
     // International ISO 8601
     // DTL  | Y| Y| Y| Y| -| M| M| -| D| D|  | H| H| :| M| M| :| S| S| .|NS|NS|NS|NS|NS|NS|NS|NS|NS
     // -----|--|--|--|--|--|--|--|--|--|--|--|--|--|--|--|--|--|--|--|--|--|--|--|--|--|--|--|--|--
     // Pos  | 1| 2| 3| 4| 5| 6| 7| 8| 9|10|11|12|13|14|15|16|17|18|19|20|21|22|23|24|25|26|27|28|29

     // Convert "Value" into "String" and place at the right position
     VAL_STRG(FORMAT := #CONVERT_FORMAT_TO_STRING,
              IN     := #date.YEAR,
              P      := #CONVERT_START_POSITION_YEAR,
              PREC   := #CONVERT_PRECISION,
              SIZE   := #CONVERT_SIZE_YEAR,
              OUT    => #tempString);    // DTL YEAR --> String --> #tempPosYear

